gs16_Sevcon2_Debug_MaxFlux				:=	USINT_TO_INT(DebugPMACControl_Rx.au8_Data[0]) +
											SHL(USINT_TO_INT(DebugPMACControl_Rx.au8_Data[1]), 8);
gs16_Sevcon2_Debug_IvLim				:=	USINT_TO_INT(DebugPMACControl_Rx.au8_Data[2]) +
											SHL(USINT_TO_INT(DebugPMACControl_Rx.au8_Data[3]), 8);
gs16_Sevcon2_Debug_IqMax				:=	USINT_TO_INT(DebugPMACControl_Rx.au8_Data[4]) +
											SHL(USINT_TO_INT(DebugPMACControl_Rx.au8_Data[5]), 8);
gs16_Sevcon2_Debug_Ls_Rx				:=	USINT_TO_INT(DebugPMACControl_Rx.au8_Data[6]) +
											SHL(USINT_TO_INT(DebugPMACControl_Rx.au8_Data[7]), 8);

gs16_Sevcon2_Debug_Slip_Rx				:=	USINT_TO_INT(DebugFVControl_Rx.au8_Data[0]) +
											SHL(USINT_TO_INT(DebugFVControl_Rx.au8_Data[1]), 8);
gs16_Sevcon2_Debug_LmSat_Rx				:=	USINT_TO_INT(DebugFVControl_Rx.au8_Data[2]) +
											SHL(USINT_TO_INT(DebugFVControl_Rx.au8_Data[3]), 8);
gs16_Sevcon2_Debug_IqMax2				:=	USINT_TO_INT(DebugFVControl_Rx.au8_Data[4]) +
											SHL(USINT_TO_INT(DebugFVControl_Rx.au8_Data[5]), 8);
gs16_Sevcon2_Debug_RecipFlux			:=	USINT_TO_INT(DebugFVControl_Rx.au8_Data[6]) +
											SHL(USINT_TO_INT(DebugFVControl_Rx.au8_Data[7]), 8);

											
TorqueStatus1_Rx_Timer(IN := NOT(TorqueStatus1_Rx.q_NewData), PT := T#3S);
TorqueStatus2_Rx_Timer(IN := NOT(TorqueStatus2_Rx.q_NewData), PT := T#3S);
TempStatus_Rx_Timer(IN := NOT(TempStatus_Rx.q_NewData), PT := T#3S);
FaultStatus_Rx_Timer(IN := NOT(FaultStatus_Rx.q_NewData), PT := T#3S);
EncoderStatus_Rx_Timer(IN := NOT(EncoderStatus_Rx.q_NewData), PT := T#3S);
DeubgCurrents_Rx_Timer(IN := NOT(DeubgCurrents_Rx.q_NewData), PT := T#3S);
DebugTemps1_Rx_Timer(IN := NOT(DebugTemps1_Rx.q_NewData), PT := T#3S);
DebugTemps2_Rx_Timer(IN := NOT(DebugTemps2_Rx.q_NewData), PT := T#3S);
DebugPMACControl_Rx_Timer(IN := NOT(DebugPMACControl_Rx.q_NewData), PT := T#3S);
DebugFVControl_Rx_Timer(IN := NOT(DebugFVControl_Rx.q_NewData), PT := T#3S);
IF (TorqueStatus1_Rx_Timer.Q = TRUE AND TorqueStatus2_Rx_Timer.Q = TRUE AND TempStatus_Rx_Timer.Q = TRUE AND
	FaultStatus_Rx_Timer.Q = TRUE AND EncoderStatus_Rx_Timer.Q = TRUE AND DeubgCurrents_Rx_Timer.Q = TRUE AND
	DebugTemps1_Rx_Timer.Q = TRUE AND DebugTemps2_Rx_Timer.Q = TRUE AND DebugPMACControl_Rx_Timer.Q = TRUE AND
	DebugFVControl_Rx_Timer.Q = TRUE) THEN
	gq_Sevcon2_CommsLoss	:=	TRUE;
ELSE
	gq_Sevcon2_CommsLoss	:=	FALSE;
END_IF											


Sevcon2_RxConversion();

END_PROGRAM

// Application/UserCode/Sevcon_Compressor/Sevcon2_RxConversion_1
PROGRAM Sevcon2_RxConversion_1
VAR
END_VAR
VAR CONSTANT
	SIXTEENTH_CF	:	REAL	:=	0.0625;
END_VAR




gr_Sevcon2_TorqueMeasured			:=	gs16_Sevcon2_TorqueMeasured_Rx * SIXTEENTH_CF;
gr_Sevcon2_TorqueAvailableForward	:=	gs16_Sevcon2_TorqueAvailableForward_Rx * SIXTEENTH_CF;
gr_Sevcon2_TorqueAvailableReverse	:=	gs16_Sevcon2_TorqueAvailableReverse_Rx * SIXTEENTH_CF;
gr_Sevcon2_DCLink_Voltage			:=	gs16_Sevcon2_DCLink_Voltage_Rx * SIXTEENTH_CF;
gr_Sevcon2_EncoderPosition			:=	LREAL_TO_REAL(gs32_Sevcon2_EncoderPosition_Rx * (1.5287890625 * EXPT(10, -5)));
gr_Sevcon2_Debug_Id_Act				:=	gs16_Sevcon2_Debug_Id_Act_Rx * SIXTEENTH_CF;
gr_Sevcon2_Debug_Iq_Act				:=	gs16_Sevcon2_Debug_Iq_Act_Rx * SIXTEENTH_CF;
gr_Sevcon2_Debug_Id_Ref				:=	gs16_Sevcon2_Debug_Id_Ref_Rx * SIXTEENTH_CF;
gr_Sevcon2_Debug_Iq_Ref				:=	gs16_Sevcon2_Debug_Iq_Ref_Rx * SIXTEENTH_CF;
gr_Sevcon2_Debug_Ls					:=	LREAL_TO_REAL(gs16_Sevcon2_Debug_Ls_Rx * (5.960464477539 * EXPT(10, -8)));
gr_Sevcon2_Debug_Slip				:=	gs16_Sevcon2_Debug_Slip_Rx * SIXTEENTH_CF;
gr_Sevcon2_Debug_LmSat				:=	LREAL_TO_REAL(gs16_Sevcon2_Debug_LmSat_Rx * (1.52587890625 * EXPT(10, -5)));

END_PROGRAM

// Application/UserCode/Sevcon_Compressor/Sevcon2_Tx_1
PROGRAM Sevcon2_Tx_1
VAR
	ht_TorqueDemand1_Tx			:	EPEC_CANVXD.Msg;
	ht_TorqueDemand2_Tx			:	EPEC_CANVXD.Msg;
	ht_BatteryDemand_Tx			:	EPEC_CANVXD.Msg;
	ht_DirectIControlDemand_Tx	:	EPEC_CANVXD.Msg;
	hton_SendTimer				:	TON;
END_VAR

Sevcon2_TxConversion();

ht_TorqueDemand1_Tx.ID		:=	16#191072FA OR EPEC_CANVXD.MASK_29BIT;
ht_TorqueDemand1_Tx.Data[0]	:=	UINT_TO_USINT(gu16_Sevcon2_TorqueRq_Tx);
ht_TorqueDemand1_Tx.Data[1]	:=	UINT_TO_USINT(SHR(gu16_Sevcon2_TorqueRq_Tx, 8));
ht_TorqueDemand1_Tx.Data[2]	:=	UINT_TO_USINT(gu16_Sevcon2_Controlword);
ht_TorqueDemand1_Tx.Data[3]	:=	UINT_TO_USINT(SHR(gu16_Sevcon2_Controlword, 8));
ht_TorqueDemand1_Tx.Data[4]	:=	UINT_TO_USINT(gu16_Sevcon2_TorqueTractionLimit_Tx);
ht_TorqueDemand1_Tx.Data[5]	:=	UINT_TO_USINT(SHR(gu16_Sevcon2_TorqueTractionLimit_Tx, 8));
ht_TorqueDemand1_Tx.Data[6]	:=	gu8_Sevcon2_SEQCommand1;
ht_TorqueDemand1_Tx.Data[7]	:=	gu8_Sevcon2_CSCommand1;
ht_TorqueDemand1_Tx.Len	:=	8;

ht_TorqueDemand2_Tx.ID		:=	16#191172FA OR EPEC_CANVXD.MASK_29BIT;
ht_TorqueDemand2_Tx.Data[0]	:=	UINT_TO_USINT(gu16_Sevcon2_TorqueRegenLimit_Tx);
ht_TorqueDemand2_Tx.Data[1]	:=	UINT_TO_USINT(SHR(gu16_Sevcon2_TorqueRegenLimit_Tx, 8));
ht_TorqueDemand2_Tx.Data[2]	:=	UINT_TO_USINT(gu16_Sevcon2_SpeedLimitForward);
ht_TorqueDemand2_Tx.Data[3]	:=	UINT_TO_USINT(SHR(gu16_Sevcon2_SpeedLimitForward, 8));
ht_TorqueDemand2_Tx.Data[4]	:=	INT_TO_USINT(gs16_Sevcon2_SpeedLimitReverse);
ht_TorqueDemand2_Tx.Data[5]	:=	INT_TO_USINT(SHR(gs16_Sevcon2_SpeedLimitReverse, 8));
ht_TorqueDemand2_Tx.Data[6]	:=	gu8_Sevcon2_SEQCommand2;
ht_TorqueDemand2_Tx.Data[7]	:=	gu8_Sevcon2_CSCommand2;
ht_TorqueDemand2_Tx.Len		:=	8;

ht_BatteryDemand_Tx.ID		:=	16#191272FA OR EPEC_CANVXD.MASK_29BIT;
ht_BatteryDemand_Tx.Data[0]	:=	UINT_TO_USINT(gu16_Sevcon2_DCLink_ImaxDischarge);
ht_BatteryDemand_Tx.Data[1]	:=	UINT_TO_USINT(SHR(gu16_Sevcon2_DCLink_ImaxDischarge, 8));
ht_BatteryDemand_Tx.Data[2]	:=	INT_TO_USINT(gs16_Sevcon2_DCLink_ImaxRecharge);
ht_BatteryDemand_Tx.Data[3]	:=	INT_TO_USINT(SHR(gs16_Sevcon2_DCLink_ImaxRecharge, 8));
ht_BatteryDemand_Tx.Data[4]	:=	UINT_TO_USINT(gu16_Sevcon2_DCLink_VoltageTarget_Tx);
ht_BatteryDemand_Tx.Data[5]	:=	UINT_TO_USINT(SHR(gu16_Sevcon2_DCLink_VoltageTarget_Tx, 8));
ht_BatteryDemand_Tx.Data[6]	:=	gu8_Sevcon1_SEQCurrentLimits;
ht_BatteryDemand_Tx.Data[7]	:=	gu8_Sevcon1_CSCurrentLimits;
ht_BatteryDemand_Tx.Len		:=	8;
	
ht_DirectIControlDemand_Tx.ID		:=	16#191372FA OR EPEC_CANVXD.MASK_29BIT;
ht_DirectIControlDemand_Tx.Data[0]	:=	UINT_TO_USINT(gu16_Sevcon2_DebugIqDirectControl_Tx);
ht_DirectIControlDemand_Tx.Data[1]	:=	UINT_TO_USINT(SHR(gu16_Sevcon2_DebugIqDirectControl_Tx, 8));
ht_DirectIControlDemand_Tx.Data[2]	:=	UINT_TO_USINT(gu16_Sevcon2_DebugIdDirectControl_Tx);
ht_DirectIControlDemand_Tx.Data[3]	:=	UINT_TO_USINT(SHR(gu16_Sevcon2_DebugIdDirectControl_Tx, 8));
ht_DirectIControlDemand_Tx.Data[4]	:=	0;
ht_DirectIControlDemand_Tx.Data[5]	:=	0;
ht_DirectIControlDemand_Tx.Data[6]	:=	gu8_Sevcon1_DirectCurrents;
ht_DirectIControlDemand_Tx.Data[7]	:=	gu8_Sevcon1_CSDirectCurrents;
ht_DirectIControlDemand_Tx.Len		:=	8;
	
hton_SendTimer(IN := TRUE, PT := T#50MS);
IF (hton_SendTimer.Q = TRUE) THEN
	G_CAN2_Channel.SendMessage(i_pMSG:=ADR(ht_TorqueDemand1_Tx));
	G_CAN2_Channel.SendMessage(i_pMSG:=ADR(ht_BatteryDemand_Tx));
	(*G_CAN2_Channel.SendMessage(i_pMSG:=ADR(ht_DirectIControlDemand_Tx));*)
	G_CAN2_Channel.SendMessage(i_pMSG:=ADR(ht_TorqueDemand2_Tx));
	hton_SendTimer(IN := FALSE, PT := T#0MS);
END_IF

END_PROGRAM

// Application/UserCode/Sevcon_Compressor/Sevcon2_TxConversion_1
PROGRAM Sevcon2_TxConversion_1
VAR
END_VAR
VAR CONSTANT
	SEVCON_TX_CF	:	REAL	:=	0.0625;
END_VAR




gu16_Sevcon2_TorqueRq_Tx				:=	REAL_TO_UINT(gr_Sevcon2_TorqueRq / SEVCON_TX_CF);
gu16_Sevcon2_TorqueTractionLimit_Tx		:=	REAL_TO_UINT(gr_Sevcon2_TorqueTractionLimit / SEVCON_TX_CF);
gu16_Sevcon2_TorqueRegenLimit_Tx		:=	REAL_TO_UINT(gr_Sevcon2_TorqueRegenLimit / SEVCON_TX_CF);
gu16_Sevcon2_DCLink_VoltageTarget_Tx	:=	REAL_TO_UINT(gr_Sevcon2_DCLink_VoltageTarget / SEVCON_TX_CF);
gu16_Sevcon2_DebugIqDirectControl_Tx	:=	REAL_TO_UINT(gr_Sevcon2_DebugIqDirectControl / SEVCON_TX_CF);
gu16_Sevcon2_DebugIdDirectControl_Tx	:=	REAL_TO_UINT(gr_Sevcon2_DebugIdDirectControl / SEVCON_TX_CF);

END_PROGRAM

// Application/UserCode/Sevcon ePTO/Sevcon_ePTO_Control
PROGRAM Sevcon_ePTO_Control
VAR_INPUT
	hton_WindUpTorque_Timer	:	TON;
	hq_PowerSteering_Enable	:	BOOL;
	hton_HandbrakeOffTimer	:	TON;
	hr_SteeringSpeed		:	REAL;
END_VAR
VAR_OUTPUT
END_VAR
VAR
	hq_ePTO_Request: BOOL := FALSE;
	hr_ePTO_Speed: INT := 400;
	gq_ePTO_Test: BOOL := FALSE;
END_VAR
VAR CONSTANT
	(*Statuswords*)
	NOTREADY_STAT				:	USINT	:=	1;
	SHUTDOWN_STAT				:	USINT	:=	2;
	PRECHARGE_STAT				:	USINT	:=	4;
	ENERGISED_STAT				:	USINT	:=	7;
	ENABLED_STAT				:	USINT	:=	8;
	FAULTREACTIONACTIVE_STAT	:	USINT	:=	11;
	FAULTOFF_STAT				:	USINT	:=	13;
	ACTIVESHORT_STAT			:	USINT	:=	14;
	(*Commandwords*)
	NOCOMMAND_COMM		:	USINT	:=	0;
	ENERGISE_COMM		:	USINT	:=	3;
	ENABLED_COMM		:	USINT	:=	5;
	SHUTDOWN_COMM		:	USINT	:=	6;
	FAULTRESET_COMM		:	USINT	:=	9;
	ACTIVESHORT_COMM	:	USINT	:=	10;
	
	TORQUE_RQ			:	USINT	:=	200;
	REVERSE_SPD_LIMIT	:	INT		:=	-500;
	MAX_DISCHARGE		:	USINT	:=	50;
	MAX_CHARGE			:	SINT	:=	-50;
	TRACTION_LIMIT		:	USINT	:=	100;
	
	CANBUS_OFF			:	INT	:=	21256;
END_VAR

VAR RETAIN
	ePTO_Speed: INT := 1200;
END_VAR



(**)
(*Check for Comms fault*)
IF (gu8_SystemState = DRIVE_SYS AND DOS_q_BatteryDischargeMain_DO = TRUE) THEN
	IF (gu8_Sevcon_ePTO_InverterStatus = FAULTOFF_STAT OR gu8_Sevcon_ePTO_InverterStatus = ACTIVESHORT_STAT) THEN
		gu16_Sevcon_ePTO_Controlword	:=	FAULTRESET_COMM;
	ELSIF (gu8_Sevcon_ePTO_InverterStatus = NOTREADY_STAT OR gu8_Sevcon_ePTO_InverterStatus = SHUTDOWN_STAT) THEN
		gu16_Sevcon_ePTO_Controlword	:=	ENERGISE_COMM;
	ELSIF (gu8_Sevcon_ePTO_InverterStatus = PRECHARGE_STAT) THEN
		gu16_Sevcon_ePTO_Controlword	:=	ENERGISE_COMM;
	ELSIF (gu8_Sevcon_ePTO_InverterStatus = ENERGISED_STAT) THEN
		gu16_Sevcon_ePTO_Controlword	:=	ENABLED_COMM;
	ELSIF (gu8_Sevcon_ePTO_InverterStatus = ENABLED_STAT) THEN
		gu16_Sevcon_ePTO_Controlword	:=	ENABLED_COMM;
	ELSE
		gu16_Sevcon_ePTO_Controlword	:=	NOCOMMAND_COMM;
	END_IF
ELSE
	gu16_Sevcon_ePTO_Controlword	:=	SHUTDOWN_COMM;
END_IF

(*hton_HandbrakeOffTimer(IN := gq_HandBrake, PT := T#30S);*)
(*This could be changed to link to the current speed of the vehicle in which case the different gear ratios and wheel diameter will be needed here to calculate*)
IF ((gq_ePTO_Test = TRUE OR DI_q_DirectionSwitch_DriveCrawl_DI = TRUE) AND gu8_SystemState = DRIVE_SYS) THEN (*change this to the input to start the body eg. oil request*)
	hq_ePTO_Request	:=	TRUE;
	hr_ePTO_Speed	:=	ePTO_Speed; (*Ensure the speed limit is never set negative*);
	gu16_Sevcon_ePTO_SpeedLimitForward	:=	REAL_TO_UINT(LIMIT(400, hr_ePTO_Speed, 2000)); (*Controlling the speed through the limits*)
	gr_Sevcon_ePTO_TorqueRq						:=	TORQUE_RQ;
ELSIF (gu8_SystemState = DRIVE_SYS) THEN
	hq_ePTO_Request	:=	FALSE;
	gu16_Sevcon_ePTO_SpeedLimitForward	:=	0;
	gr_Sevcon_ePTO_TorqueRq				:=	0;
END_IF



(*All these are constants to be sent out to the Sevcon unit and do not need changing during operation*)
(*IF (gu8_Sevcon_ePTO_InverterStatus = ENABLED_STAT) THEN
	hton_WindUpTorque_Timer(IN := TRUE, PT := T#5000MS);
	gr_Sevcon_ePTO_TorqueRq						:=	TORQUE_RQ * (TIME_TO_REAL(hton_WindUpTorque_Timer.ET) / 5000);
ELSE
	hton_WindUpTorque_Timer(IN := FALSE, PT := T#0MS);
	gr_Sevcon_ePTO_TorqueRq						:=	0;
END_IF*)

gr_Sevcon_ePTO_DCLink_VoltageTarget			:=	0; (*Not needed as not being used as a generator*)
gs16_Sevcon_ePTO_SpeedLimitReverse			:=	REVERSE_SPD_LIMIT;
gu16_Sevcon_ePTO_DCLink_ImaxDischarge		:=	MAX_DISCHARGE;
gs16_Sevcon_ePTO_DCLink_ImaxRecharge		:=	MAX_CHARGE;
gr_Sevcon_ePTO_TorqueTractionLimit			:=	TRACTION_LIMIT;
gr_Sevcon_ePTO_TorqueRegenLimit				:=	0;

gu8_Sevcon_ePTO_CSCommand1					:=	0;
gu8_Sevcon_ePTO_CSCommand2					:=	0;
gu8_Sevcon_ePTO_CSCurrentLimits				:=	0;
(*Counters to run every cycle and increment so the Sevcons know the VMU is still running*)
IF (gu8_Sevcon_ePTO_SEQCommand1 < 255) THEN
	gu8_Sevcon_ePTO_SEQCommand1			:=	gu8_Sevcon_ePTO_SEQCommand1 + 1;
ELSE
	gu8_Sevcon_ePTO_SEQCommand1			:=	0;
END_IF
IF (gu8_Sevcon_ePTO_SEQCommand2 < 255) THEN
	gu8_Sevcon_ePTO_SEQCommand2			:=	gu8_Sevcon_ePTO_SEQCommand2 + 1;
ELSE
	gu8_Sevcon_ePTO_SEQCommand2			:=	0;
END_IF
IF (gu8_Sevcon_ePTO_SEQCurrentLimits < 255) THEN
	gu8_Sevcon_ePTO_SEQCurrentLimits	:=	gu8_Sevcon_ePTO_SEQCurrentLimits + 1;
ELSE
	gu8_Sevcon_ePTO_SEQCurrentLimits	:=	0;
END_IF

END_PROGRAM

// Application/UserCode/Sevcon ePTO/Sevcon_ePTO_Rx
PROGRAM Sevcon_ePTO_Rx
VAR
	TorqueStatus1_Rx	:	Receive_CAN4_EXD;
	TorqueStatus2_Rx	:	Receive_CAN4_EXD;
	TempStatus_Rx		:	Receive_CAN4_EXD;
	FaultStatus_Rx		:	Receive_CAN4_EXD;
	EncoderStatus_Rx	:	Receive_CAN4_EXD;
	DeubgCurrents_Rx	:	Receive_CAN4_EXD;
	DebugTemps1_Rx		:	Receive_CAN4_EXD;
	DebugTemps2_Rx		:	Receive_CAN4_EXD;
	DebugPMACControl_Rx	:	Receive_CAN4_EXD;
	DebugFVControl_Rx	:	Receive_CAN4_EXD;
END_VAR


TorqueStatus1_Rx(u32_COBID	:=	16#1918FF73,
				q_NewData => ,
				au8_Data => ,
				u8_Length => 			);

TorqueStatus2_Rx(u32_COBID	:=	16#1919FF73,
				q_NewData => ,
				au8_Data => ,
				u8_Length => 			);

TempStatus_Rx(u32_COBID	:=	16#191AFF73,
				q_NewData => ,
				au8_Data => ,
				u8_Length => 			);

FaultStatus_Rx(u32_COBID	:=	16#191BFF73,
				q_NewData => ,
				au8_Data => ,
				u8_Length => 			);

EncoderStatus_Rx(u32_COBID	:=	16#191CFF73,
				q_NewData => ,
				au8_Data => ,
				u8_Length => 			);

DeubgCurrents_Rx(u32_COBID	:=	16#1928FF73,
				q_NewData => ,
				au8_Data => ,
				u8_Length => 			);

DebugTemps1_Rx(u32_COBID	:=	16#192AFF73,
				q_NewData => ,
				au8_Data => ,
				u8_Length => 			);

DebugTemps2_Rx(u32_COBID	:=	16#192BFF73,
				q_NewData => ,
				au8_Data => ,
				u8_Length => 			);

DebugPMACControl_Rx(u32_COBID	:=	16#192CFF73,
				q_NewData => ,
				au8_Data => ,
				u8_Length => 			);

DebugFVControl_Rx(u32_COBID	:=	16#192DFF73,
				q_NewData => ,
				au8_Data => ,
				u8_Length => 			);				

			
				
gs16_Sevcon_ePTO_TorqueMeasured_Rx			:=	USINT_TO_INT(TorqueStatus1_Rx.au8_Data[0]) +
											SHL(USINT_TO_INT(TorqueStatus1_Rx.au8_Data[1]), 8);
gs16_Sevcon_ePTO_SpeedMeasured				:=	USINT_TO_INT(TorqueStatus1_Rx.au8_Data[2]) +
											SHL(USINT_TO_INT(TorqueStatus1_Rx.au8_Data[3]), 8);
gs16_Sevcon_ePTO_DCLink_Current				:=	USINT_TO_INT(TorqueStatus1_Rx.au8_Data[4]) +
											SHL(USINT_TO_INT(TorqueStatus1_Rx.au8_Data[5]), 8);
gu8_Sevcon_ePTO_SEQ_Torque					:=	TorqueStatus1_Rx.au8_Data[6];
gu8_Sevcon_ePTO_CS_Torque					:=	TorqueStatus1_Rx.au8_Data[7];

gs16_Sevcon_ePTO_TorqueAvailableForward_Rx	:=	USINT_TO_INT(TorqueStatus2_Rx.au8_Data[0]) +
											SHL(USINT_TO_INT(TorqueStatus2_Rx.au8_Data[1]), 8);
gs16_Sevcon_ePTO_TorqueAvailableReverse_Rx	:=	USINT_TO_INT(TorqueStatus2_Rx.au8_Data[2]) +
											SHL(USINT_TO_INT(TorqueStatus2_Rx.au8_Data[3]), 8);
gu8_Sevcon_ePTO_InverterStatus				:=	TorqueStatus2_Rx.au8_Data[4];
gu8_Sevcon_ePTO_TorqueLimitCode				:=	TorqueStatus2_Rx.au8_Data[5];
gu8_Sevcon_ePTO_SEQ_Status					:=	TorqueStatus2_Rx.au8_Data[6];
gu8_Sevcon_ePTO_CS_Status					:=	TorqueStatus2_Rx.au8_Data[7];

gs16_Sevcon_ePTO_TempRemaining				:=	USINT_TO_INT(TempStatus_Rx.au8_Data[0]) +
											SHL(USINT_TO_INT(TempStatus_Rx.au8_Data[1]), 8);
gs16_Sevcon_ePTO_MotorTemp					:=	USINT_TO_INT(TempStatus_Rx.au8_Data[2]) +
											SHL(USINT_TO_INT(TempStatus_Rx.au8_Data[3]), 8);
gs16_Sevcon_ePTO_DCLink_Voltage_Rx			:=	USINT_TO_INT(TempStatus_Rx.au8_Data[4]) +
											SHL(USINT_TO_INT(TempStatus_Rx.au8_Data[5]), 8);
gu8_Sevcon_ePTO_SEQ_Temp					:=	TempStatus_Rx.au8_Data[6];
gu8_Sevcon_ePTO_CS_Temp						:=	TempStatus_Rx.au8_Data[7];

gs16_Sevcon_ePTO_FaultCode					:=	USINT_TO_INT(FaultStatus_Rx.au8_Data[0]) +
											SHL(USINT_TO_INT(FaultStatus_Rx.au8_Data[1]), 8);
gs32_Sevcon_ePTO_FaultData					:=	USINT_TO_DINT(FaultStatus_Rx.au8_Data[2]) +
											SHL(USINT_TO_DINT(FaultStatus_Rx.au8_Data[3]), 8) +
											SHL(USINT_TO_DINT(FaultStatus_Rx.au8_Data[4]), 16) +
											SHL(USINT_TO_DINT(FaultStatus_Rx.au8_Data[5]), 24);
gu8_Sevcon_ePTO_SEQ_Fault					:=	FaultStatus_Rx.au8_Data[6];
gu8_Sevcon_ePTO_CS_Fault					:=	FaultStatus_Rx.au8_Data[7];

gs32_Sevcon_ePTO_EncoderPosition_Rx			:=	USINT_TO_DINT(EncoderStatus_Rx.au8_Data[0]) +
											SHL(USINT_TO_DINT(EncoderStatus_Rx.au8_Data[1]), 8) +
											SHL(USINT_TO_DINT(EncoderStatus_Rx.au8_Data[2]), 16) +
											SHL(USINT_TO_DINT(EncoderStatus_Rx.au8_Data[3]), 24);

gs16_Sevcon_ePTO_Debug_Id_Act_Rx			:=	USINT_TO_INT(DeubgCurrents_Rx.au8_Data[0]) +
											SHL(USINT_TO_INT(DeubgCurrents_Rx.au8_Data[1]), 8);
gs16_Sevcon_ePTO_Debug_Iq_Act_Rx			:=	USINT_TO_INT(DeubgCurrents_Rx.au8_Data[2]) +
											SHL(USINT_TO_INT(DeubgCurrents_Rx.au8_Data[3]), 8);
gs16_Sevcon_ePTO_Debug_Id_Ref_Rx			:=	USINT_TO_INT(DeubgCurrents_Rx.au8_Data[4]) +
											SHL(USINT_TO_INT(DeubgCurrents_Rx.au8_Data[5]), 8);
gs16_Sevcon_ePTO_Debug_Iq_Ref_Rx			:=	USINT_TO_INT(DeubgCurrents_Rx.au8_Data[6]) +
											SHL(USINT_TO_INT(DeubgCurrents_Rx.au8_Data[7]), 8);

gu8_Sevcon_ePTO_Debug_Temp_Junction0		:=	DebugTemps1_Rx.au8_Data[0];
gu8_Sevcon_ePTO_Debug_Temp_Junction1		:=	DebugTemps1_Rx.au8_Data[1];
gu8_Sevcon_ePTO_Debug_Temp_Junction2		:=	DebugTemps1_Rx.au8_Data[2];
gu8_Sevcon_ePTO_Debug_Temp_Junction3		:=	DebugTemps1_Rx.au8_Data[3];
gu8_Sevcon_ePTO_Debug_Temp_Junction4		:=	DebugTemps1_Rx.au8_Data[4];
gu8_Sevcon_ePTO_Debug_Temp_Junction5		:=	DebugTemps1_Rx.au8_Data[5];
gu8_Sevcon_ePTO_Debug_Temp_MotorMeasured	:=	DebugTemps1_Rx.au8_Data[6];
gu8_Sevcon_ePTO_Debug_Temp_MotorEstimate	:=	DebugTemps1_Rx.au8_Data[7];

gu8_Sevcon_ePTO_Debug_Temp_CapEstimateFast	:=	DebugTemps2_Rx.au8_Data[0];
gu8_Sevcon_ePTO_Debug_Temp_Track			:=	DebugTemps2_Rx.au8_Data[1];
gu8_Sevcon_ePTO_Debug_Temp_CapEstimateSlow	:=	DebugTemps2_Rx.au8_Data[2];
gu8_Sevcon_ePTO_Debug_Temp_Heatsink			:=	DebugTemps2_Rx.au8_Data[3];
gu8_Sevcon_ePTO_Debug_Temp_DeltaTj			:=	DebugTemps2_Rx.au8_Data[4];
gu8_Sevcon_ePTO_Debug_Temp_Normalised		:=	DebugTemps2_Rx.au8_Data[5];
gu8_Sevcon_ePTO_Debug_Temp_Coolant			:=	DebugTemps2_Rx.au8_Data[6];
gu8_Sevcon_ePTO_Debug_Temp_Winding			:=	DebugTemps2_Rx.au8_Data[7];

gs16_Sevcon_ePTO_Debug_MaxFlux				:=	USINT_TO_INT(DebugPMACControl_Rx.au8_Data[0]) +
											SHL(USINT_TO_INT(DebugPMACControl_Rx.au8_Data[1]), 8);
gs16_Sevcon_ePTO_Debug_IvLim				:=	USINT_TO_INT(DebugPMACControl_Rx.au8_Data[2]) +
											SHL(USINT_TO_INT(DebugPMACControl_Rx.au8_Data[3]), 8);
gs16_Sevcon_ePTO_Debug_IqMax				:=	USINT_TO_INT(DebugPMACControl_Rx.au8_Data[4]) +
											SHL(USINT_TO_INT(DebugPMACControl_Rx.au8_Data[5]), 8);
gs16_Sevcon_ePTO_Debug_Ls_Rx				:=	USINT_TO_INT(DebugPMACControl_Rx.au8_Data[6]) +
											SHL(USINT_TO_INT(DebugPMACControl_Rx.au8_Data[7]), 8);

gs16_Sevcon_ePTO_Debug_Slip_Rx				:=	USINT_TO_INT(DebugFVControl_Rx.au8_Data[0]) +
											SHL(USINT_TO_INT(DebugFVControl_Rx.au8_Data[1]), 8);
gs16_Sevcon_ePTO_Debug_LmSat_Rx				:=	USINT_TO_INT(DebugFVControl_Rx.au8_Data[2]) +
											SHL(USINT_TO_INT(DebugFVControl_Rx.au8_Data[3]), 8);
gs16_Sevcon_ePTO_Debug_IqMax2				:=	USINT_TO_INT(DebugFVControl_Rx.au8_Data[4]) +
											SHL(USINT_TO_INT(DebugFVControl_Rx.au8_Data[5]), 8);
gs16_Sevcon_ePTO_Debug_RecipFlux			:=	USINT_TO_INT(DebugFVControl_Rx.au8_Data[6]) +
											SHL(USINT_TO_INT(DebugFVControl_Rx.au8_Data[7]), 8);


											
Sevcon_ePTO_RxConversion();

END_PROGRAM

// Application/UserCode/Sevcon ePTO/Sevcon_ePTO_RxConversion
PROGRAM Sevcon_ePTO_RxConversion
VAR
END_VAR
VAR CONSTANT
	SIXTEENTH_CF	:	REAL	:=	0.0625;
END_VAR




gr_Sevcon_ePTO_TorqueMeasured			:=	gs16_Sevcon_ePTO_TorqueMeasured_Rx * SIXTEENTH_CF;
gr_Sevcon_ePTO_TorqueAvailableForward	:=	gs16_Sevcon_ePTO_TorqueAvailableForward_Rx * SIXTEENTH_CF;
gr_Sevcon_ePTO_TorqueAvailableReverse	:=	gs16_Sevcon_ePTO_TorqueAvailableReverse_Rx * SIXTEENTH_CF;
gr_Sevcon_ePTO_DCLink_Voltage			:=	gs16_Sevcon_ePTO_DCLink_Voltage_Rx * SIXTEENTH_CF;
gr_Sevcon_ePTO_EncoderPosition			:=	LREAL_TO_REAL(gs32_Sevcon_ePTO_EncoderPosition_Rx * (1.5287890625 * EXPT(10, -5)));
gr_Sevcon_ePTO_Debug_Id_Act			:=	gs16_Sevcon_ePTO_Debug_Id_Act_Rx * SIXTEENTH_CF;
gr_Sevcon_ePTO_Debug_Iq_Act			:=	gs16_Sevcon_ePTO_Debug_Iq_Act_Rx * SIXTEENTH_CF;
gr_Sevcon_ePTO_Debug_Id_Ref			:=	gs16_Sevcon_ePTO_Debug_Id_Ref_Rx * SIXTEENTH_CF;
gr_Sevcon_ePTO_Debug_Iq_Ref			:=	gs16_Sevcon_ePTO_Debug_Iq_Ref_Rx * SIXTEENTH_CF;
gr_Sevcon_ePTO_Debug_Ls				:=	LREAL_TO_REAL(gs16_Sevcon_ePTO_Debug_Ls_Rx * (5.960464477539 * EXPT(10, -8)));
gr_Sevcon_ePTO_Debug_Slip				:=	gs16_Sevcon_ePTO_Debug_Slip_Rx * SIXTEENTH_CF;
gr_Sevcon_ePTO_Debug_LmSat				:=	LREAL_TO_REAL(gs16_Sevcon_ePTO_Debug_LmSat_Rx * (1.52587890625 * EXPT(10, -5)));

END_PROGRAM

// Application/UserCode/Sevcon ePTO/Sevcon_ePTO_Tx
PROGRAM Sevcon_ePTO_Tx
VAR
	ht_TorqueDemand1_Tx			:	EPEC_CANVXD.Msg;
	ht_TorqueDemand2_Tx			:	EPEC_CANVXD.Msg;
	ht_BatteryDemand_Tx			:	EPEC_CANVXD.Msg;
	ht_DirectIControlDemand_Tx	:	EPEC_CANVXD.Msg;
	hton_SendTimer				:	TON;
END_VAR

Sevcon_ePTO_TxConversion();

ht_TorqueDemand1_Tx.ID		:=	16#191073FA (*191071FA*) OR EPEC_CANVXD.MASK_29BIT;
ht_TorqueDemand1_Tx.Data[0]	:=	UINT_TO_USINT(gu16_Sevcon_ePTO_TorqueRq_Tx);
ht_TorqueDemand1_Tx.Data[1]	:=	UINT_TO_USINT(SHR(gu16_Sevcon_ePTO_TorqueRq_Tx, 8));
ht_TorqueDemand1_Tx.Data[2]	:=	UINT_TO_USINT(gu16_Sevcon_ePTO_Controlword);
ht_TorqueDemand1_Tx.Data[3]	:=	UINT_TO_USINT(SHR(gu16_Sevcon_ePTO_Controlword, 8));
ht_TorqueDemand1_Tx.Data[4]	:=	UINT_TO_USINT(gu16_Sevcon_ePTO_TorqueTractionLimit_Tx);
ht_TorqueDemand1_Tx.Data[5]	:=	UINT_TO_USINT(SHR(gu16_Sevcon_ePTO_TorqueTractionLimit_Tx, 8));
ht_TorqueDemand1_Tx.Data[6]	:=	gu8_Sevcon_ePTO_SEQCommand1;
ht_TorqueDemand1_Tx.Data[7]	:=	gu8_Sevcon_ePTO_CSCommand1;
ht_TorqueDemand1_Tx.Len	:=	8;

ht_TorqueDemand2_Tx.ID		:=	16#191173FA (*191171FA*) OR EPEC_CANVXD.MASK_29BIT;
ht_TorqueDemand2_Tx.Data[0]	:=	UINT_TO_USINT(gu16_Sevcon_ePTO_TorqueRegenLimit_Tx);
ht_TorqueDemand2_Tx.Data[1]	:=	UINT_TO_USINT(SHR(gu16_Sevcon_ePTO_TorqueRegenLimit_Tx, 8));
ht_TorqueDemand2_Tx.Data[2]	:=	UINT_TO_USINT(gu16_Sevcon_ePTO_SpeedLimitForward);
ht_TorqueDemand2_Tx.Data[3]	:=	UINT_TO_USINT(SHR(gu16_Sevcon_ePTO_SpeedLimitForward, 8));
ht_TorqueDemand2_Tx.Data[4]	:=	INT_TO_USINT(gs16_Sevcon_ePTO_SpeedLimitReverse);
ht_TorqueDemand2_Tx.Data[5]	:=	INT_TO_USINT(SHR(gs16_Sevcon_ePTO_SpeedLimitReverse, 8));
ht_TorqueDemand2_Tx.Data[6]	:=	gu8_Sevcon_ePTO_SEQCommand2;
ht_TorqueDemand2_Tx.Data[7]	:=	gu8_Sevcon_ePTO_CSCommand2;
ht_TorqueDemand2_Tx.Len		:=	8;

ht_BatteryDemand_Tx.ID		:=	16#191273FA (*191271FA*) OR EPEC_CANVXD.MASK_29BIT;
ht_BatteryDemand_Tx.Data[0]	:=	UINT_TO_USINT(gu16_Sevcon_ePTO_DCLink_ImaxDischarge);
ht_BatteryDemand_Tx.Data[1]	:=	UINT_TO_USINT(SHR(gu16_Sevcon_ePTO_DCLink_ImaxDischarge, 8));
ht_BatteryDemand_Tx.Data[2]	:=	INT_TO_USINT(gs16_Sevcon_ePTO_DCLink_ImaxRecharge);
ht_BatteryDemand_Tx.Data[3]	:=	INT_TO_USINT(SHR(gs16_Sevcon_ePTO_DCLink_ImaxRecharge, 8));
ht_BatteryDemand_Tx.Data[4]	:=	UINT_TO_USINT(gu16_Sevcon_ePTO_DCLink_VoltageTarget_Tx);
ht_BatteryDemand_Tx.Data[5]	:=	UINT_TO_USINT(SHR(gu16_Sevcon_ePTO_DCLink_VoltageTarget_Tx, 8));
ht_BatteryDemand_Tx.Data[6]	:=	gu8_Sevcon_ePTO_SEQCurrentLimits;
ht_BatteryDemand_Tx.Data[7]	:=	gu8_Sevcon_ePTO_CSCurrentLimits;
ht_BatteryDemand_Tx.Len		:=	8;
	
ht_DirectIControlDemand_Tx.ID		:=	16#191373FA (*191371FA*) OR EPEC_CANVXD.MASK_29BIT;
ht_DirectIControlDemand_Tx.Data[0]	:=	UINT_TO_USINT(gu16_Sevcon_ePTO_DebugIqDirectControl_Tx);
ht_DirectIControlDemand_Tx.Data[1]	:=	UINT_TO_USINT(SHR(gu16_Sevcon_ePTO_DebugIqDirectControl_Tx, 8));
ht_DirectIControlDemand_Tx.Data[2]	:=	UINT_TO_USINT(gu16_Sevcon_ePTO_DebugIdDirectControl_Tx);
ht_DirectIControlDemand_Tx.Data[3]	:=	UINT_TO_USINT(SHR(gu16_Sevcon_ePTO_DebugIdDirectControl_Tx, 8));
ht_DirectIControlDemand_Tx.Data[4]	:=	0;
ht_DirectIControlDemand_Tx.Data[5]	:=	0;
ht_DirectIControlDemand_Tx.Data[6]	:=	gu8_Sevcon_ePTO_DirectCurrents;
ht_DirectIControlDemand_Tx.Data[7]	:=	gu8_Sevcon_ePTO_CSDirectCurrents;
ht_DirectIControlDemand_Tx.Len		:=	8;
	
hton_SendTimer(IN := TRUE, PT := T#50MS);
IF (hton_SendTimer.Q = TRUE) THEN
	G_CAN4_Channel.SendMessage(i_pMSG:=ADR(ht_TorqueDemand1_Tx));
	G_CAN4_Channel.SendMessage(i_pMSG:=ADR(ht_BatteryDemand_Tx));
	G_CAN4_Channel.SendMessage(i_pMSG:=ADR(ht_DirectIControlDemand_Tx));
	G_CAN4_Channel.SendMessage(i_pMSG:=ADR(ht_TorqueDemand2_Tx));
	hton_SendTimer(IN := FALSE, PT := T#0MS);
END_IF

END_PROGRAM

// Application/UserCode/Sevcon ePTO/Sevcon_ePTO_TxConversion
PROGRAM Sevcon_ePTO_TxConversion
VAR
END_VAR
VAR CONSTANT
	SEVCON_TX_CF	:	REAL	:=	0.0625;
END_VAR




gu16_Sevcon_ePTO_TorqueRq_Tx				:=	REAL_TO_UINT(gr_Sevcon_ePTO_TorqueRq / SEVCON_TX_CF);
gu16_Sevcon_ePTO_TorqueTractionLimit_Tx		:=	REAL_TO_UINT(gr_Sevcon_ePTO_TorqueTractionLimit / SEVCON_TX_CF);
gu16_Sevcon_ePTO_TorqueRegenLimit_Tx		:=	REAL_TO_UINT(gr_Sevcon_ePTO_TorqueRegenLimit / SEVCON_TX_CF);
gu16_Sevcon_ePTO_DCLink_VoltageTarget_Tx	:=	REAL_TO_UINT(gr_Sevcon_ePTO_DCLink_VoltageTarget / SEVCON_TX_CF);
gu16_Sevcon_ePTO_DebugIqDirectControl_Tx	:=	REAL_TO_UINT(gr_Sevcon_ePTO_DebugIqDirectControl / SEVCON_TX_CF);
gu16_Sevcon_ePTO_DebugIdDirectControl_Tx	:=	REAL_TO_UINT(gr_Sevcon_ePTO_DebugIdDirectControl / SEVCON_TX_CF);

END_PROGRAM

// Application/UserCode/Sevcon_PSP/Sevcon_Steer_Control_1
PROGRAM Sevcon_Steer_Control_1
VAR
	hton_WindUpTorque_Timer	:	TON;
	hq_PowerSteering_Enable	:	BOOL;
	hton_HandbrakeOffTimer	:	TON;
	hr_SteeringSpeed		:	REAL;
	hton_PowerSteeringOff	:	TON;
	Steering_Speed_Setpoint: INT := 2200; //changed from 2000
END_VAR
VAR CONSTANT
	(*Statuswords*)
	NOTREADY_STAT				:	USINT	:=	1;
	SHUTDOWN_STAT				:	USINT	:=	2;
	PRECHARGE_STAT				:	USINT	:=	4;
	ENERGISED_STAT				:	USINT	:=	7;
	ENABLED_STAT				:	USINT	:=	8;
	FAULTREACTIONACTIVE_STAT	:	USINT	:=	11;
	FAULTOFF_STAT				:	USINT	:=	13;
	ACTIVESHORT_STAT			:	USINT	:=	14;
	(*Commandwords*)
	NOCOMMAND_COMM		:	USINT	:=	0;
	ENERGISE_COMM		:	USINT	:=	3;
	ENABLED_COMM		:	USINT	:=	5;
	SHUTDOWN_COMM		:	USINT	:=	6;
	FAULTRESET_COMM		:	USINT	:=	9;
	ACTIVESHORT_COMM	:	USINT	:=	10;
	
	TORQUE_RQ			:	USINT	:=	200;
	REVERSE_SPD_LIMIT	:	INT		:=	-500;
	MAX_DISCHARGE		:	USINT	:=	50;
	MAX_CHARGE			:	SINT	:=	-50;
	TRACTION_LIMIT		:	USINT	:=	100;
	
	CANBUS_OFF			:	INT	:=	21256;
END_VAR


(**)
(*Check for Comms fault*)
IF (gu8_SystemState = DRIVE_SYS AND DOS_q_BatteryDischargeMain_DO = TRUE) THEN
	DO_q_DrievtrainPowerSteering_DO	:=	TRUE;
	IF (gu8_Sevcon1_InverterStatus = FAULTOFF_STAT OR gu8_Sevcon1_InverterStatus = ACTIVESHORT_STAT) THEN
		gu16_Sevcon1_Controlword	:=	FAULTRESET_COMM;
	ELSIF (gu8_Sevcon1_InverterStatus = NOTREADY_STAT OR gu8_Sevcon1_InverterStatus = SHUTDOWN_STAT) THEN
		gu16_Sevcon1_Controlword	:=	ENERGISE_COMM;
	ELSIF (gu8_Sevcon1_InverterStatus = PRECHARGE_STAT) THEN
		gu16_Sevcon1_Controlword	:=	ENERGISE_COMM;
	ELSIF (gu8_Sevcon1_InverterStatus = ENERGISED_STAT) THEN
		gu16_Sevcon1_Controlword	:=	ENABLED_COMM;
	ELSIF (gu8_Sevcon1_InverterStatus = ENABLED_STAT) THEN
		gu16_Sevcon1_Controlword	:=	ENABLED_COMM;
	ELSE
		gu16_Sevcon1_Controlword	:=	NOCOMMAND_COMM;
	END_IF
ELSE
	DO_q_DrievtrainPowerSteering_DO	:=	FALSE;
	gu16_Sevcon1_Controlword	:=	SHUTDOWN_COMM;
END_IF

hton_HandbrakeOffTimer(IN := HMI_Rx.Hand_Brake_On, PT := T#10MS); //Time changed from 30s to 10ms

(*This could be changed to link to the current speed of the vehicle in which case the different gear ratios and wheel diameter will be needed here to calculate*)
IF ((HMI_Rx.Hand_Brake_On = FALSE OR NOT gq_Gear_Neutral) AND gu8_SystemState = DRIVE_SYS) THEN //TEST FIRST THEN REMOVE THIS COMMENT OR NOT gq_Gear_Neutral
	hq_PowerSteering_Enable	:=	TRUE;
	hr_SteeringSpeed		:=	MAX(REAL_TO_INT(Steering_Speed_Setpoint - (ABS(gr_VehicleSpeed_kmph) * 10)), 0) (*Ensure the speed limit is never set negative*);
	gu16_Sevcon1_SpeedLimitForward	:=	REAL_TO_UINT(LIMIT(200, hr_SteeringSpeed, Steering_Speed_Setpoint)); (*Controlling the speed through the limits*)
	hton_PowerSteeringOff(IN := FALSE, PT := T#0S);
ELSIF ((hton_HandbrakeOffTimer.Q = TRUE AND ABS(gr_VehicleSpeed_kmph) < 3) AND gu8_SystemState = DRIVE_SYS) THEN //AND before DRIVE_SYS changed from OR
	hq_PowerSteering_Enable	:=	FALSE;
	hton_PowerSteeringOff(IN := TRUE, PT := T#10MS);
	
	IF (hton_PowerSteeringOff.Q = TRUE) THEN
		gu16_Sevcon1_SpeedLimitForward	:=	200; //instead of shutting off reduce speed to a minimum
	ELSE
		gu16_Sevcon1_SpeedLimitForward	:=	650;
	END_IF
	
END_IF


(*All these are constants to be sent out to the Sevcon unit and do not need changing during operation*)
IF (gu8_Sevcon1_InverterStatus = ENABLED_STAT) THEN
	hton_WindUpTorque_Timer(IN := TRUE, PT := T#5000MS);
	gr_Sevcon1_TorqueRq						:=	TORQUE_RQ * (TIME_TO_REAL(hton_WindUpTorque_Timer.ET) / 5000);
ELSE
	hton_WindUpTorque_Timer(IN := FALSE, PT := T#0MS);
	gr_Sevcon1_TorqueRq						:=	0;
END_IF

gr_Sevcon1_DCLink_VoltageTarget			:=	0; (*Not needed as not being used as a generator*)
gs16_Sevcon1_SpeedLimitReverse			:=	REVERSE_SPD_LIMIT;
gu16_Sevcon1_DCLink_ImaxDischarge		:=	MAX_DISCHARGE;
gs16_Sevcon1_DCLink_ImaxRecharge		:=	MAX_CHARGE;
gr_Sevcon1_TorqueTractionLimit			:=	TRACTION_LIMIT;
gr_Sevcon1_TorqueRegenLimit				:=	0;

gu8_Sevcon1_CSCommand1					:=	0;
gu8_Sevcon1_CSCommand2					:=	0;
gu8_Sevcon1_CSCurrentLimits				:=	0;

(*Counters to run every cycle and increment so the Sevcons know the VMU is still running*)
IF (gu8_Sevcon1_SEQCommand1 < 255) THEN
	gu8_Sevcon1_SEQCommand1			:=	gu8_Sevcon1_SEQCommand1 + 1;
ELSE
	gu8_Sevcon1_SEQCommand1			:=	0;
END_IF
IF (gu8_Sevcon1_SEQCommand2 < 255) THEN
	gu8_Sevcon1_SEQCommand2			:=	gu8_Sevcon1_SEQCommand2 + 1;
ELSE
	gu8_Sevcon1_SEQCommand2			:=	0;
END_IF
IF (gu8_Sevcon1_SEQCurrentLimits < 255) THEN
	gu8_Sevcon1_SEQCurrentLimits	:=	gu8_Sevcon1_SEQCurrentLimits + 1;
ELSE
	gu8_Sevcon1_SEQCurrentLimits	:=	0;
END_IF

(*Backup Pump*)
IF (hq_PowerSteering_Enable = TRUE AND gs16_Sevcon1_FaultCode = CANBUS_OFF) THEN (* Matt, does something else need ORed*)
	DO_q_BackupPump_DO	:=	TRUE;
	(*Fault state will set from the sevcon error*)
ELSE
	DO_q_BackupPump_DO	:=	FALSE;
END_IF

END_PROGRAM

// Application/UserCode/Sevcon_PSP/Sevcon_Steer_Rx_1
PROGRAM Sevcon_Steer_Rx_1
VAR
	TorqueStatus1_Rx	:	Receive_CAN2_EXD;
	TorqueStatus2_Rx	:	Receive_CAN2_EXD;
	TempStatus_Rx		:	Receive_CAN2_EXD;
	FaultStatus_Rx		:	Receive_CAN2_EXD;
	EncoderStatus_Rx	:	Receive_CAN2_EXD;
	DeubgCurrents_Rx	:	Receive_CAN2_EXD;
	DebugTemps1_Rx		:	Receive_CAN2_EXD;
	DebugTemps2_Rx		:	Receive_CAN2_EXD;
	DebugPMACControl_Rx	:	Receive_CAN2_EXD;
	DebugFVControl_Rx	:	Receive_CAN2_EXD;
	
	TorqueStatus1_Rx_Timer		:	TON;
	TorqueStatus2_Rx_Timer		:	TON;
	TempStatus_Rx_Timer			:	TON;
	FaultStatus_Rx_Timer		:	TON;
	EncoderStatus_Rx_Timer		:	TON;
	DeubgCurrents_Rx_Timer		:	TON;
	DebugTemps1_Rx_Timer		:	TON;
	DebugTemps2_Rx_Timer		:	TON;
	DebugPMACControl_Rx_Timer	:	TON;
	DebugFVControl_Rx_Timer		:	TON;
END_VAR


TorqueStatus1_Rx(u32_COBID	:=	16#1918FF71,
				q_NewData => ,
				au8_Data => ,
				u8_Length => 			);

TorqueStatus2_Rx(u32_COBID	:=	16#1919FF71,
				q_NewData => ,
				au8_Data => ,
				u8_Length => 			);

TempStatus_Rx(u32_COBID	:=	16#191AFF71,
				q_NewData => ,
				au8_Data => ,
				u8_Length => 			);

FaultStatus_Rx(u32_COBID	:=	16#191BFF71,
				q_NewData => ,
				au8_Data => ,
				u8_Length => 			);

EncoderStatus_Rx(u32_COBID	:=	16#191CFF71,
				q_NewData => ,
				au8_Data => ,
				u8_Length => 			);

DeubgCurrents_Rx(u32_COBID	:=	16#1928FF71,
				q_NewData => ,
				au8_Data => ,
				u8_Length => 			);

DebugTemps1_Rx(u32_COBID	:=	16#192AFF71,
				q_NewData => ,
				au8_Data => ,
				u8_Length => 			);

DebugTemps2_Rx(u32_COBID	:=	16#192BFF71,
				q_NewData => ,
				au8_Data => ,
				u8_Length => 			);

DebugPMACControl_Rx(u32_COBID	:=	16#192CFF71,
				q_NewData => ,
				au8_Data => ,
				u8_Length => 			);

DebugFVControl_Rx(u32_COBID	:=	16#192DFF71,
				q_NewData => ,
				au8_Data => ,
				u8_Length => 			);				

			
				
gs16_Sevcon1_TorqueMeasured_Rx			:=	USINT_TO_INT(TorqueStatus1_Rx.au8_Data[0]) +
											SHL(USINT_TO_INT(TorqueStatus1_Rx.au8_Data[1]), 8);
gs16_Sevcon1_SpeedMeasured				:=	USINT_TO_INT(TorqueStatus1_Rx.au8_Data[2]) +
											SHL(USINT_TO_INT(TorqueStatus1_Rx.au8_Data[3]), 8);
gs16_Sevcon1_DCLink_Current				:=	USINT_TO_INT(TorqueStatus1_Rx.au8_Data[4]) +
											SHL(USINT_TO_INT(TorqueStatus1_Rx.au8_Data[5]), 8);
gu8_Sevcon1_SEQ_Torque					:=	TorqueStatus1_Rx.au8_Data[6];
gu8_Sevcon1_CS_Torque					:=	TorqueStatus1_Rx.au8_Data[7];

gs16_Sevcon1_TorqueAvailableForward_Rx	:=	USINT_TO_INT(TorqueStatus2_Rx.au8_Data[0]) +
											SHL(USINT_TO_INT(TorqueStatus2_Rx.au8_Data[1]), 8);
gs16_Sevcon1_TorqueAvailableReverse_Rx	:=	USINT_TO_INT(TorqueStatus2_Rx.au8_Data[2]) +
											SHL(USINT_TO_INT(TorqueStatus2_Rx.au8_Data[3]), 8);
gu8_Sevcon1_InverterStatus				:=	TorqueStatus2_Rx.au8_Data[4];
gu8_Sevcon1_TorqueLimitCode				:=	TorqueStatus2_Rx.au8_Data[5];
gu8_Sevcon1_SEQ_Status					:=	TorqueStatus2_Rx.au8_Data[6];
gu8_Sevcon1_CS_Status					:=	TorqueStatus2_Rx.au8_Data[7];

gs16_Sevcon1_TempRemaining				:=	USINT_TO_INT(TempStatus_Rx.au8_Data[0]) +
											SHL(USINT_TO_INT(TempStatus_Rx.au8_Data[1]), 8);
gs16_Sevcon1_MotorTemp					:=	USINT_TO_INT(TempStatus_Rx.au8_Data[2]) +
											SHL(USINT_TO_INT(TempStatus_Rx.au8_Data[3]), 8);
gs16_Sevcon1_DCLink_Voltage_Rx			:=	USINT_TO_INT(TempStatus_Rx.au8_Data[4]) +
											SHL(USINT_TO_INT(TempStatus_Rx.au8_Data[5]), 8);
gu8_Sevcon1_SEQ_Temp					:=	TempStatus_Rx.au8_Data[6];
gu8_Sevcon1_CS_Temp						:=	TempStatus_Rx.au8_Data[7];

gs16_Sevcon1_FaultCode					:=	USINT_TO_INT(FaultStatus_Rx.au8_Data[0]) +
											SHL(USINT_TO_INT(FaultStatus_Rx.au8_Data[1]), 8);
gs32_Sevcon1_FaultData					:=	USINT_TO_DINT(FaultStatus_Rx.au8_Data[2]) +
											SHL(USINT_TO_DINT(FaultStatus_Rx.au8_Data[3]), 8) +
											SHL(USINT_TO_DINT(FaultStatus_Rx.au8_Data[4]), 16) +
											SHL(USINT_TO_DINT(FaultStatus_Rx.au8_Data[5]), 24);
gu8_Sevcon1_SEQ_Fault					:=	FaultStatus_Rx.au8_Data[6];
gu8_Sevcon1_CS_Fault					:=	FaultStatus_Rx.au8_Data[7];

gs32_Sevcon1_EncoderPosition_Rx			:=	USINT_TO_DINT(EncoderStatus_Rx.au8_Data[0]) +
											SHL(USINT_TO_DINT(EncoderStatus_Rx.au8_Data[1]), 8) +
											SHL(USINT_TO_DINT(EncoderStatus_Rx.au8_Data[2]), 16) +
											SHL(USINT_TO_DINT(EncoderStatus_Rx.au8_Data[3]), 24);

gs16_Sevcon1_Debug_Id_Act_Rx			:=	USINT_TO_INT(DeubgCurrents_Rx.au8_Data[0]) +
											SHL(USINT_TO_INT(DeubgCurrents_Rx.au8_Data[1]), 8);
gs16_Sevcon1_Debug_Iq_Act_Rx			:=	USINT_TO_INT(DeubgCurrents_Rx.au8_Data[2]) +
											SHL(USINT_TO_INT(DeubgCurrents_Rx.au8_Data[3]), 8);
gs16_Sevcon1_Debug_Id_Ref_Rx			:=	USINT_TO_INT(DeubgCurrents_Rx.au8_Data[4]) +
											SHL(USINT_TO_INT(DeubgCurrents_Rx.au8_Data[5]), 8);
gs16_Sevcon1_Debug_Iq_Ref_Rx			:=	USINT_TO_INT(DeubgCurrents_Rx.au8_Data[6]) +
											SHL(USINT_TO_INT(DeubgCurrents_Rx.au8_Data[7]), 8);

gu8_Sevcon1_Debug_Temp_Junction0		:=	DebugTemps1_Rx.au8_Data[0];
gu8_Sevcon1_Debug_Temp_Junction1		:=	DebugTemps1_Rx.au8_Data[1];
gu8_Sevcon1_Debug_Temp_Junction2		:=	DebugTemps1_Rx.au8_Data[2];
gu8_Sevcon1_Debug_Temp_Junction3		:=	DebugTemps1_Rx.au8_Data[3];
gu8_Sevcon1_Debug_Temp_Junction4		:=	DebugTemps1_Rx.au8_Data[4];
gu8_Sevcon1_Debug_Temp_Junction5		:=	DebugTemps1_Rx.au8_Data[5];
gu8_Sevcon1_Debug_Temp_MotorMeasured	:=	DebugTemps1_Rx.au8_Data[6];
gu8_Sevcon1_Debug_Temp_MotorEstimate	:=	DebugTemps1_Rx.au8_Data[7];

gu8_Sevcon1_Debug_Temp_CapEstimateFast	:=	DebugTemps2_Rx.au8_Data[0];
gu8_Sevcon1_Debug_Temp_Track			:=	DebugTemps2_Rx.au8_Data[1];
gu8_Sevcon1_Debug_Temp_CapEstimateSlow	:=	DebugTemps2_Rx.au8_Data[2];
gu8_Sevcon1_Debug_Temp_Heatsink			:=	DebugTemps2_Rx.au8_Data[3];
gu8_Sevcon1_Debug_Temp_DeltaTj			:=	DebugTemps2_Rx.au8_Data[4];
gu8_Sevcon1_Debug_Temp_Normalised		:=	DebugTemps2_Rx.au8_Data[5];
gu8_Sevcon1_Debug_Temp_Coolant			:=	DebugTemps2_Rx.au8_Data[6];
gu8_Sevcon1_Debug_Temp_Winding			:=	DebugTemps2_Rx.au8_Data[7];

gs16_Sevcon1_Debug_MaxFlux				:=	USINT_TO_INT(DebugPMACControl_Rx.au8_Data[0]) +
											SHL(USINT_TO_INT(DebugPMACControl_Rx.au8_Data[1]), 8);
gs16_Sevcon1_Debug_IvLim				:=	USINT_TO_INT(DebugPMACControl_Rx.au8_Data[2]) +
											SHL(USINT_TO_INT(DebugPMACControl_Rx.au8_Data[3]), 8);
gs16_Sevcon1_Debug_IqMax				:=	USINT_TO_INT(DebugPMACControl_Rx.au8_Data[4]) +
											SHL(USINT_TO_INT(DebugPMACControl_Rx.au8_Data[5]), 8);
gs16_Sevcon1_Debug_Ls_Rx				:=	USINT_TO_INT(DebugPMACControl_Rx.au8_Data[6]) +
											SHL(USINT_TO_INT(DebugPMACControl_Rx.au8_Data[7]), 8);

gs16_Sevcon1_Debug_Slip_Rx				:=	USINT_TO_INT(DebugFVControl_Rx.au8_Data[0]) +
											SHL(USINT_TO_INT(DebugFVControl_Rx.au8_Data[1]), 8);
gs16_Sevcon1_Debug_LmSat_Rx				:=	USINT_TO_INT(DebugFVControl_Rx.au8_Data[2]) +
											SHL(USINT_TO_INT(DebugFVControl_Rx.au8_Data[3]), 8);
gs16_Sevcon1_Debug_IqMax2				:=	USINT_TO_INT(DebugFVControl_Rx.au8_Data[4]) +
											SHL(USINT_TO_INT(DebugFVControl_Rx.au8_Data[5]), 8);
gs16_Sevcon1_Debug_RecipFlux			:=	USINT_TO_INT(DebugFVControl_Rx.au8_Data[6]) +
											SHL(USINT_TO_INT(DebugFVControl_Rx.au8_Data[7]), 8);


TorqueStatus1_Rx_Timer(IN := NOT(TorqueStatus1_Rx.q_NewData), PT := T#3S);
TorqueStatus2_Rx_Timer(IN := NOT(TorqueStatus2_Rx.q_NewData), PT := T#3S);
TempStatus_Rx_Timer(IN := NOT(TempStatus_Rx.q_NewData), PT := T#3S);
FaultStatus_Rx_Timer(IN := NOT(FaultStatus_Rx.q_NewData), PT := T#3S);
EncoderStatus_Rx_Timer(IN := NOT(EncoderStatus_Rx.q_NewData), PT := T#3S);
DeubgCurrents_Rx_Timer(IN := NOT(DeubgCurrents_Rx.q_NewData), PT := T#3S);
DebugTemps1_Rx_Timer(IN := NOT(DebugTemps1_Rx.q_NewData), PT := T#3S);
DebugTemps2_Rx_Timer(IN := NOT(DebugTemps2_Rx.q_NewData), PT := T#3S);
DebugPMACControl_Rx_Timer(IN := NOT(DebugPMACControl_Rx.q_NewData), PT := T#3S);
DebugFVControl_Rx_Timer(IN := NOT(DebugFVControl_Rx.q_NewData), PT := T#3S);
IF (TorqueStatus1_Rx_Timer.Q = TRUE AND TorqueStatus2_Rx_Timer.Q = TRUE AND TempStatus_Rx_Timer.Q = TRUE AND
	FaultStatus_Rx_Timer.Q = TRUE AND EncoderStatus_Rx_Timer.Q = TRUE AND DeubgCurrents_Rx_Timer.Q = TRUE AND
	DebugTemps1_Rx_Timer.Q = TRUE AND DebugTemps2_Rx_Timer.Q = TRUE AND DebugPMACControl_Rx_Timer.Q = TRUE AND
	DebugFVControl_Rx_Timer.Q = TRUE) THEN
	gq_Sevcon1_CommsLoss	:=	TRUE;
ELSE
	gq_Sevcon1_CommsLoss	:=	FALSE;
END_IF
										
Sevcon_Steer_RxConversion();

END_PROGRAM

// Application/UserCode/Sevcon_PSP/Sevcon_Steer_RxConversion_1
PROGRAM Sevcon_Steer_RxConversion_1
VAR
END_VAR
VAR CONSTANT
	SIXTEENTH_CF	:	REAL	:=	0.0625;
END_VAR




gr_Sevcon1_TorqueMeasured			:=	gs16_Sevcon1_TorqueMeasured_Rx * SIXTEENTH_CF;
gr_Sevcon1_TorqueAvailableForward	:=	gs16_Sevcon1_TorqueAvailableForward_Rx * SIXTEENTH_CF;
gr_Sevcon1_TorqueAvailableReverse	:=	gs16_Sevcon1_TorqueAvailableReverse_Rx * SIXTEENTH_CF;
gr_Sevcon1_DCLink_Voltage			:=	gs16_Sevcon1_DCLink_Voltage_Rx * SIXTEENTH_CF;
gr_Sevcon1_EncoderPosition			:=	LREAL_TO_REAL(gs32_Sevcon1_EncoderPosition_Rx * (1.5287890625 * EXPT(10, -5)));
gr_Sevcon1_Debug_Id_Act				:=	gs16_Sevcon1_Debug_Id_Act_Rx * SIXTEENTH_CF;
gr_Sevcon1_Debug_Iq_Act				:=	gs16_Sevcon1_Debug_Iq_Act_Rx * SIXTEENTH_CF;
gr_Sevcon1_Debug_Id_Ref				:=	gs16_Sevcon1_Debug_Id_Ref_Rx * SIXTEENTH_CF;
gr_Sevcon1_Debug_Iq_Ref				:=	gs16_Sevcon1_Debug_Iq_Ref_Rx * SIXTEENTH_CF;
gr_Sevcon1_Debug_Ls					:=	LREAL_TO_REAL(gs16_Sevcon1_Debug_Ls_Rx * (5.960464477539 * EXPT(10, -8)));
gr_Sevcon1_Debug_Slip				:=	gs16_Sevcon1_Debug_Slip_Rx * SIXTEENTH_CF;
gr_Sevcon1_Debug_LmSat				:=	LREAL_TO_REAL(gs16_Sevcon1_Debug_LmSat_Rx * (1.52587890625 * EXPT(10, -5)));

END_PROGRAM

// Application/UserCode/Sevcon_PSP/Sevcon_Steer_Tx_1
PROGRAM Sevcon_Steer_Tx_1
VAR
	ht_TorqueDemand1_Tx			:	EPEC_CANVXD.Msg;
	ht_TorqueDemand2_Tx			:	EPEC_CANVXD.Msg;
	ht_BatteryDemand_Tx			:	EPEC_CANVXD.Msg;
	ht_DirectIControlDemand_Tx	:	EPEC_CANVXD.Msg;
	hton_SendTimer				:	TON;
END_VAR

Sevcon_Steer_TxConversion();

ht_TorqueDemand1_Tx.ID		:=	16#191071FA OR EPEC_CANVXD.MASK_29BIT;
ht_TorqueDemand1_Tx.Data[0]	:=	UINT_TO_USINT(gu16_Sevcon1_TorqueRq_Tx);
ht_TorqueDemand1_Tx.Data[1]	:=	UINT_TO_USINT(SHR(gu16_Sevcon1_TorqueRq_Tx, 8));
ht_TorqueDemand1_Tx.Data[2]	:=	UINT_TO_USINT(gu16_Sevcon1_Controlword);
ht_TorqueDemand1_Tx.Data[3]	:=	UINT_TO_USINT(SHR(gu16_Sevcon1_Controlword, 8));
ht_TorqueDemand1_Tx.Data[4]	:=	UINT_TO_USINT(gu16_Sevcon1_TorqueTractionLimit_Tx);
ht_TorqueDemand1_Tx.Data[5]	:=	UINT_TO_USINT(SHR(gu16_Sevcon1_TorqueTractionLimit_Tx, 8));
ht_TorqueDemand1_Tx.Data[6]	:=	gu8_Sevcon1_SEQCommand1;
ht_TorqueDemand1_Tx.Data[7]	:=	gu8_Sevcon1_CSCommand1;
ht_TorqueDemand1_Tx.Len	:=	8;

ht_TorqueDemand2_Tx.ID		:=	16#191171FA OR EPEC_CANVXD.MASK_29BIT;
ht_TorqueDemand2_Tx.Data[0]	:=	UINT_TO_USINT(gu16_Sevcon1_TorqueRegenLimit_Tx);
ht_TorqueDemand2_Tx.Data[1]	:=	UINT_TO_USINT(SHR(gu16_Sevcon1_TorqueRegenLimit_Tx, 8));
ht_TorqueDemand2_Tx.Data[2]	:=	UINT_TO_USINT(gu16_Sevcon1_SpeedLimitForward);
ht_TorqueDemand2_Tx.Data[3]	:=	UINT_TO_USINT(SHR(gu16_Sevcon1_SpeedLimitForward, 8));
ht_TorqueDemand2_Tx.Data[4]	:=	INT_TO_USINT(gs16_Sevcon1_SpeedLimitReverse);
ht_TorqueDemand2_Tx.Data[5]	:=	INT_TO_USINT(SHR(gs16_Sevcon1_SpeedLimitReverse, 8));
ht_TorqueDemand2_Tx.Data[6]	:=	gu8_Sevcon1_SEQCommand2;
ht_TorqueDemand2_Tx.Data[7]	:=	gu8_Sevcon1_CSCommand2;
ht_TorqueDemand2_Tx.Len		:=	8;

ht_BatteryDemand_Tx.ID		:=	16#191271FA OR EPEC_CANVXD.MASK_29BIT;
ht_BatteryDemand_Tx.Data[0]	:=	UINT_TO_USINT(gu16_Sevcon1_DCLink_ImaxDischarge);
ht_BatteryDemand_Tx.Data[1]	:=	UINT_TO_USINT(SHR(gu16_Sevcon1_DCLink_ImaxDischarge, 8));
ht_BatteryDemand_Tx.Data[2]	:=	INT_TO_USINT(gs16_Sevcon1_DCLink_ImaxRecharge);
ht_BatteryDemand_Tx.Data[3]	:=	INT_TO_USINT(SHR(gs16_Sevcon1_DCLink_ImaxRecharge, 8));
ht_BatteryDemand_Tx.Data[4]	:=	UINT_TO_USINT(gu16_Sevcon1_DCLink_VoltageTarget_Tx);
ht_BatteryDemand_Tx.Data[5]	:=	UINT_TO_USINT(SHR(gu16_Sevcon1_DCLink_VoltageTarget_Tx, 8));
ht_BatteryDemand_Tx.Data[6]	:=	gu8_Sevcon1_SEQCurrentLimits;
ht_BatteryDemand_Tx.Data[7]	:=	gu8_Sevcon1_CSCurrentLimits;
ht_BatteryDemand_Tx.Len		:=	8;
	
ht_DirectIControlDemand_Tx.ID		:=	16#191371FA OR EPEC_CANVXD.MASK_29BIT;
ht_DirectIControlDemand_Tx.Data[0]	:=	UINT_TO_USINT(gu16_Sevcon1_DebugIqDirectControl_Tx);
ht_DirectIControlDemand_Tx.Data[1]	:=	UINT_TO_USINT(SHR(gu16_Sevcon1_DebugIqDirectControl_Tx, 8));
ht_DirectIControlDemand_Tx.Data[2]	:=	UINT_TO_USINT(gu16_Sevcon1_DebugIdDirectControl_Tx);
ht_DirectIControlDemand_Tx.Data[3]	:=	UINT_TO_USINT(SHR(gu16_Sevcon1_DebugIdDirectControl_Tx, 8));
ht_DirectIControlDemand_Tx.Data[4]	:=	0;
ht_DirectIControlDemand_Tx.Data[5]	:=	0;
ht_DirectIControlDemand_Tx.Data[6]	:=	gu8_Sevcon1_DirectCurrents;
ht_DirectIControlDemand_Tx.Data[7]	:=	gu8_Sevcon1_CSDirectCurrents;
ht_DirectIControlDemand_Tx.Len		:=	8;
	
hton_SendTimer(IN := TRUE, PT := T#50MS);
IF (hton_SendTimer.Q = TRUE) THEN
	G_CAN2_Channel.SendMessage(i_pMSG:=ADR(ht_TorqueDemand1_Tx));
	G_CAN2_Channel.SendMessage(i_pMSG:=ADR(ht_BatteryDemand_Tx));
	G_CAN2_Channel.SendMessage(i_pMSG:=ADR(ht_DirectIControlDemand_Tx));
	G_CAN2_Channel.SendMessage(i_pMSG:=ADR(ht_TorqueDemand2_Tx));
	hton_SendTimer(IN := FALSE, PT := T#0MS);
END_IF

END_PROGRAM

// Application/UserCode/Sevcon_PSP/Sevcon_Steer_TxConversion_1
PROGRAM Sevcon_Steer_TxConversion_1
VAR
END_VAR
VAR CONSTANT
	SEVCON_TX_CF	:	REAL	:=	0.0625;
END_VAR




gu16_Sevcon1_TorqueRq_Tx				:=	REAL_TO_UINT(gr_Sevcon1_TorqueRq / SEVCON_TX_CF);
gu16_Sevcon1_TorqueTractionLimit_Tx		:=	REAL_TO_UINT(gr_Sevcon1_TorqueTractionLimit / SEVCON_TX_CF);
gu16_Sevcon1_TorqueRegenLimit_Tx		:=	REAL_TO_UINT(gr_Sevcon1_TorqueRegenLimit / SEVCON_TX_CF);
gu16_Sevcon1_DCLink_VoltageTarget_Tx	:=	REAL_TO_UINT(gr_Sevcon1_DCLink_VoltageTarget / SEVCON_TX_CF);
gu16_Sevcon1_DebugIqDirectControl_Tx	:=	REAL_TO_UINT(gr_Sevcon1_DebugIqDirectControl / SEVCON_TX_CF);
gu16_Sevcon1_DebugIdDirectControl_Tx	:=	REAL_TO_UINT(gr_Sevcon1_DebugIdDirectControl / SEVCON_TX_CF);

END_PROGRAM

// Application/UserCode/BMS/CATL/CATLBMS_RxConversion
PROGRAM CATLBMS_RxConversion

(*Convert input variables into real units by applying conversion factors and offsets*)

END_PROGRAM

// Application/UserCode/BMS/CATL/CATLBMS1_Rx_1
PROGRAM CATLBMS1_Rx_1

(*Program to receive all data from the CATL BMS*)



(*Initial saving CAN messages to receipt strucutres*)


(*Unpacking structures into variables*)


(*Comms loss check to ensure all messages are still being received*)


CATLBMS_RxConversion();

END_PROGRAM

// Application/UserCode/BMS/CATL/CATLBMS_RxConversion_1
PROGRAM CATLBMS_RxConversion_1

(*Convert input variables into real units by applying conversion factors and offsets*)

END_PROGRAM

// Application/UserCode/BMS/OrionBMS/Orion_Control_1
PROGRAM Orion_Control_1
VAR
	OrionPause_Timer	:	TON;
	hton_DisconnectionPause_Timer	:	TON;
END_VAR

(*Program to control the BMS during operation*)
(*Setting battery mode*)
IF (gu8_SystemState = DRIVE_SYS) THEN
	(*Have an initial short pause after contactors have closed before changing into discharge mode*)
	OrionPause_Timer(IN := TRUE, PT := T#20mS);
	IF (OrionPause_Timer.Q = TRUE) THEN
		(*Set discharge output*)
		DO_q_DrivetrainKL15C_DO	:=	FALSE;
		DO_q_DrivetrainKL15D_DO	:=	TRUE;
		(*Request on CAN the BMS into operational mode*)
		gu8_BMS1_MPO_1_State	:=	1;
		gu8_BMS1_MPO_2_State	:=	1; (* This does F_ALL *)
		gu8_BMS2_MPO_1_State	:=	1;
		gu8_BMS2_MPO_2_State	:=	1;
		
		
	END_IF
	hton_DisconnectionPause_Timer(IN := FALSE, PT := T#0MS);
ELSIF (gu8_SystemState = PLUGIN_SYS) THEN
	(*Have an initial short pause after contactors have closed before changing into charge mode*)
	OrionPause_Timer(IN := TRUE, PT := T#20MS);
	IF (OrionPause_Timer.Q = TRUE) THEN
		(*Set outputs for charge mode*)
		DO_q_DrivetrainKL15C_DO	:=	TRUE;
		DO_q_DrivetrainKL15D_DO	:=	FALSE;
		(*Request on CAN the BMS into operational mode*)
		gu8_BMS1_MPO_1_State	:=	0;
		gu8_BMS1_MPO_2_State	:=	0;
		gu8_BMS2_MPO_1_State	:=	0;
		gu8_BMS2_MPO_2_State	:=	0;
	END_IF
	hton_DisconnectionPause_Timer(IN := FALSE, PT := T#0MS);
ELSIF (DO_q_BatteryDischargeMain_DO = FALSE AND DO_q_Battery1ChargeMain_DO = FALSE AND DO_q_Battery2ChargeMain_DO = FALSE AND
		DO_q_BatteryDischargePrecharge_DO = FALSE AND DO_q_Battery1ChargePrecharge_DO = FALSE AND DO_q_Battery2ChargePrecharge_DO = FALSE) THEN
	(*Only perform disconnect of batteries when all contactors are opened to prevent them from damaging their own contactors Explain ??MAT *)
	hton_DisconnectionPause_Timer(IN := TRUE, PT := T#100MS);
	IF (hton_DisconnectionPause_Timer.Q = TRUE) THEN
		DO_q_DrivetrainKL15C_DO	:=	FALSE;
		DO_q_DrivetrainKL15D_DO	:=	FALSE;
		(*Request the BMS inactive*)
		gu8_BMS1_MPO_1_State	:=	0;
		gu8_BMS1_MPO_2_State	:=	0;
		gu8_BMS2_MPO_1_State	:=	0;
		gu8_BMS2_MPO_2_State	:=	0;
			
	END_IF
	OrionPause_Timer(IN := FALSE, PT := t#0ms);
END_IF
IF HMI_Rx.PB_BMS1_DTC_Reset THEN
	gu8_BMS1_MPO_3_State :=1;
	ELSE gu8_BMS1_MPO_3_State :=0;
END_IF
IF HMI_Rx.PB_BMS2_DTC_Reset THEN
	gu8_BMS2_MPO_3_State :=1;
	ELSE gu8_BMS2_MPO_3_State :=0;
END_IF

END_PROGRAM

// Application/UserCode/BMS/OrionBMS/OrionBMS1_Rx_1
PROGRAM OrionBMS1_Rx_1
VAR
	OrionBMS1_6B0_Rx	:	Receive_CAN2_STD;
	OrionBMS1_6B1_Rx	:	Receive_CAN2_STD;
	OrionBMS1_6B2_Rx	:	Receive_CAN2_STD;
	OrionBMS1_6B3_Rx	:	Receive_CAN2_STD;
	OrionBMS1_6B4_Rx	:	Receive_CAN2_STD;
	OrionBMS1_6B5_Rx	:	Receive_CAN2_STD;
	OrionBMS1_6B6_Rx	:	Receive_CAN2_STD;
	OrionBMS1_6B7_Rx	:	Receive_CAN2_STD;
	OrionBMS1_6B8_Rx	:	Receive_CAN2_STD;
	OrionBMS1_6B9_Rx	:	Receive_CAN2_STD;
	OrionBMS1_6BA_Rx	:	Receive_CAN2_STD;
	OrionBMS1_6BB_Rx	:	Receive_CAN2_STD;
	OrionBMS1_6BC_Rx	:	Receive_CAN2_STD;
	OrionBMS1_6BD_Rx	:	Receive_CAN2_STD;
	
	OrionBMS1_6B0_Rx_Timer	:	TON;
	OrionBMS1_6B1_Rx_Timer	:	TON;
	OrionBMS1_6B2_Rx_Timer	:	TON;
	OrionBMS1_6B3_Rx_Timer	:	TON;
	OrionBMS1_6B4_Rx_Timer	:	TON;
	OrionBMS1_6B5_Rx_Timer	:	TON;
	OrionBMS1_6B6_Rx_Timer	:	TON;
	OrionBMS1_6B7_Rx_Timer	:	TON;
	OrionBMS1_6B8_Rx_Timer	:	TON;
	OrionBMS1_6B9_Rx_Timer	:	TON;
	OrionBMS1_6BA_Rx_Timer	:	TON;
	OrionBMS1_6BB_Rx_Timer	:	TON;
	OrionBMS1_6BC_Rx_Timer	:	TON;
	OrionBMS1_6BD_Rx_Timer	:	TON;
	END_VAR

(*Program to receive all data from the Orion BMS*)
(*Initial saving CAN messages to receipt strucutres*)
OrionBMS1_6B0_Rx(u32_COBID	:=	16#6B0,
				 q_NewData => ,
				 au8_Data => ,
				 u8_Length => 			);
				 
OrionBMS1_6B1_Rx(u32_COBID	:=	16#6B1,
				 q_NewData => ,
				 au8_Data => ,
				 u8_Length => 			);
				 
OrionBMS1_6B2_Rx(u32_COBID	:=	16#6B2,
				 q_NewData => ,
				 au8_Data => ,
				 u8_Length => 			);
				 
OrionBMS1_6B3_Rx(u32_COBID	:=	16#6B3,
				 q_NewData => ,
				 au8_Data => ,
				 u8_Length => 			);
				 
OrionBMS1_6B4_Rx(u32_COBID	:=	16#6B4,
				 q_NewData => ,
				 au8_Data => ,
				 u8_Length => 			);
				 
OrionBMS1_6B5_Rx(u32_COBID	:=	16#6B5,
				 q_NewData => ,
				 au8_Data => ,
				 u8_Length => 			);
				 
OrionBMS1_6B6_Rx(u32_COBID	:=	16#6B6,
				 q_NewData => ,
				 au8_Data => ,
				 u8_Length => 			);
				 
OrionBMS1_6B7_Rx(u32_COBID	:=	16#6B7,
				 q_NewData => ,
				 au8_Data => ,
				 u8_Length => 			);
			 
OrionBMS1_6B8_Rx(u32_COBID	:=	16#6B8,
				 q_NewData => ,
				 au8_Data => ,
				 u8_Length => 			);
				 
OrionBMS1_6B9_Rx(u32_COBID	:=	16#6B9,
				 q_NewData => ,
				 au8_Data => ,
				 u8_Length => 			);
				 
OrionBMS1_6BA_Rx(u32_COBID	:=	16#6BA,
				 q_NewData => ,
				 au8_Data => ,
				 u8_Length => 			);
				 
OrionBMS1_6BB_Rx(u32_COBID	:=	16#6BB,
				 q_NewData => ,
				 au8_Data => ,
				 u8_Length => 			);
				 
OrionBMS1_6BC_Rx(u32_COBID	:=	16#6BC,
				 q_NewData => ,
				 au8_Data => ,
				 u8_Length => 			);
				 
OrionBMS1_6BD_Rx(u32_COBID	:=	16#6BD,
				 q_NewData => ,
				 au8_Data => ,
				 u8_Length => 			);


(*Unpacking structures into variables*)
(*6B0*)
gs16_OrionBMS1_PackCurrent	:=	USINT_TO_INT(OrionBMS1_6B0_Rx.au8_Data[0]) +
								SHL(USINT_TO_INT(OrionBMS1_6B0_Rx.au8_Data[1]), 8);
gu16_OrionBMS1_RAW_Pack_Voltage	:=	USINT_TO_UINT(OrionBMS1_6B0_Rx.au8_Data[2]) +
								SHL(USINT_TO_UINT(OrionBMS1_6B0_Rx.au8_Data[3]), 8);
gu8_OrionBMS1_RAW_SOC	:=	OrionBMS1_6B0_Rx.au8_Data[4];
gu16_OrionBMS1_RelayState	:=	USINT_TO_UINT(OrionBMS1_6B0_Rx.au8_Data[5]) +
								SHL(USINT_TO_UINT(OrionBMS1_6B0_Rx.au8_Data[6]), 8);
gu8_OrionBMS1_Custom_Flag_1	:=	OrionBMS1_6B0_Rx.au8_Data[7];

(*6B1*)
gu8_OrionBMS1_Isolation_ADC			:=	USINT_TO_UINT(OrionBMS1_6B1_Rx.au8_Data[0]) +
									SHL(USINT_TO_UINT(OrionBMS1_6B1_Rx.au8_Data[1]), 8);
gu8_OrionBMS1_Shortest_Wave			:=	USINT_TO_UINT(OrionBMS1_6B1_Rx.au8_Data[2]) +
									SHL(USINT_TO_UINT(OrionBMS1_6B1_Rx.au8_Data[3]), 8);
gu16_OrionBMS1_Isolation_Clipping	:=	USINT_TO_UINT(OrionBMS1_6B1_Rx.au8_Data[4]) +
									SHL(USINT_TO_UINT(OrionBMS1_6B1_Rx.au8_Data[5]), 8);
gu16_OrionBMS1_Isolation_Threshold	:=	USINT_TO_UINT(OrionBMS1_6B1_Rx.au8_Data[6]) +
									SHL(USINT_TO_UINT(OrionBMS1_6B1_Rx.au8_Data[7]), 8);
									
(*6B2*)
gu16_OrionBMS1_DTC_Flags1		:=	USINT_TO_UINT(OrionBMS1_6B2_Rx.au8_Data[0]) +
								SHL(USINT_TO_UINT(OrionBMS1_6B2_Rx.au8_Data[1]), 8);
gu16_OrionBMS1_DTC_Flags2		:=	USINT_TO_UINT(OrionBMS1_6B2_Rx.au8_Data[2]) +
								SHL(USINT_TO_UINT(OrionBMS1_6B2_Rx.au8_Data[3]), 8);
gu16_OrionBMS1_FailsafeStatus	:=	USINT_TO_UINT(OrionBMS1_6B2_Rx.au8_Data[4]) +
								SHL(USINT_TO_UINT(OrionBMS1_6B2_Rx.au8_Data[5]), 8);
gu16_OrionBMS1_Current_Limit_Status		:=	USINT_TO_UINT(OrionBMS1_6B2_Rx.au8_Data[6]) +
								SHL(USINT_TO_UINT(OrionBMS1_6B2_Rx.au8_Data[7]), 8);
(*6B3*)
gu8_OrionBMS1_PackHealth			:=	OrionBMS1_6B3_Rx.au8_Data[0];
gu16_OrionBMS1_PackCycles			:=	USINT_TO_UINT(OrionBMS1_6B3_Rx.au8_Data[1]) +
									SHL(USINT_TO_UINT(OrionBMS1_6B3_Rx.au8_Data[2]), 8);
gu16_OrionBMS1_PackResistance		:=	USINT_TO_UINT(OrionBMS1_6B3_Rx.au8_Data[3]) +
									SHL(USINT_TO_UINT(OrionBMS1_6B3_Rx.au8_Data[4]), 8);
gu8_OrionBMS1_PopulatedCells		:=	OrionBMS1_6B3_Rx.au8_Data[5];
gu16_OrionBMS1_MaximumPackVoltage	:=	USINT_TO_UINT (OrionBMS1_6B3_Rx.au8_Data[6]) +
									SHL(USINT_TO_UINT(OrionBMS1_6B3_Rx.au8_Data[7]),8);

(*6B4*)
gu8_OrionBMS1_HighTemp		:=	OrionBMS1_6B4_Rx.au8_Data[0];
gu8_OrionBMS1_LowTemp		:=	OrionBMS1_6B4_Rx.au8_Data[1];
gu8_OrionBMS1_AverageTemp	:=	OrionBMS1_6B4_Rx.au8_Data[2];
gu8_OrionBMS1_InternalTemp	:=	OrionBMS1_6B4_Rx.au8_Data[3];
gu16_OrionBMS1_MinimumPackVoltage	:=	USINT_TO_UINT(OrionBMS1_6B4_Rx.au8_Data[4]) +
									SHL(USINT_TO_UINT(OrionBMS1_6B4_Rx.au8_Data[5]), 8);
gu16_OrionBMS1_PackAmphours	:=	USINT_TO_UINT(OrionBMS1_6B4_Rx.au8_Data[6]) +
								SHL(USINT_TO_UINT(OrionBMS1_6B4_Rx.au8_Data[7]), 8);
(*6B5*)
gu16_OrionBMS1_AverageCellVoltage	:=	USINT_TO_UINT(OrionBMS1_6B5_Rx.au8_Data[0]) +
										SHL(USINT_TO_UINT(OrionBMS1_6B5_Rx.au8_Data[1]), 8);
gu16_OrionBMS1_LowCellVoltage		:=	USINT_TO_UINT(OrionBMS1_6B5_Rx.au8_Data[2]) +
										SHL(USINT_TO_UINT(OrionBMS1_6B5_Rx.au8_Data[3]), 8);
gu16_OrionBMS1_HighCellVoltage		:=	USINT_TO_UINT(OrionBMS1_6B5_Rx.au8_Data[4]) +
										SHL(USINT_TO_UINT(OrionBMS1_6B5_Rx.au8_Data[5]), 8);
gu8_OrionBMS1_LowCellVoltNumber		:=	OrionBMS1_6B5_Rx.au8_Data[6];
gu8_OrionBMS1_HighCellVoltNumber	:=	OrionBMS1_6B5_Rx.au8_Data[7];
(*6B6*)
gu8_OrionBMS1_Low_Intres_ID			:=	OrionBMS1_6B6_Rx.au8_Data[0];
gu8_OrionBMS1_High_Intres_ID		:=	OrionBMS1_6B6_Rx.au8_Data[1];
gu16_OrionBMS1_Low_Cell_Resistance	:=	USINT_TO_UINT(OrionBMS1_6B6_Rx.au8_Data[2]) +
										SHL(USINT_TO_UINT(OrionBMS1_6B6_Rx.au8_Data[3]), 8);
gu16_OrionBMS1_High_Cell_Resistance	:=	USINT_TO_UINT(OrionBMS1_6B6_Rx.au8_Data[4]) +
										SHL(USINT_TO_UINT(OrionBMS1_6B6_Rx.au8_Data[5]), 8);
gu16_OrionBMS1_Average_Cell_Resistance	:=	USINT_TO_UINT(OrionBMS1_6B6_Rx.au8_Data[6]) +
										SHL(USINT_TO_UINT(OrionBMS1_6B6_Rx.au8_Data[7]), 8);

(*6B7*)
gu8_OrionBMS1_Low_Thermistor_ID			:=	OrionBMS1_6B7_Rx.au8_Data[0];
gu8_OrionBMS1_High_Thermistor_ID		:=	OrionBMS1_6B7_Rx.au8_Data[1];
gu16_OrionBMS1_PackDCL				:=	USINT_TO_UINT(OrionBMS1_6B7_Rx.au8_Data[2]) +
										SHL(USINT_TO_UINT(OrionBMS1_6B7_Rx.au8_Data[3]), 8);
gu16_OrionBMS1_PackCCL				:=	USINT_TO_UINT(OrionBMS1_6B7_Rx.au8_Data[4]) +
										SHL(USINT_TO_UINT(OrionBMS1_6B7_Rx.au8_Data[5]), 8);
gu16_OrionBMS1_PackSummedVoltage	:=	USINT_TO_UINT(OrionBMS1_6B7_Rx.au8_Data[6]) +
										SHL(USINT_TO_UINT(OrionBMS1_6B7_Rx.au8_Data[7]), 8);

(*6B8*)
	gu8_OrionBMS1_Firmware_Minor		:=	OrionBMS1_6B8_Rx.au8_Data[0];	
	gu8_OrionBMS1_Firmware_Patch		:=	OrionBMS1_6B8_Rx.au8_Data[1];		
	gu8_OrionBMS1_Constant_2			:=	OrionBMS1_6B8_Rx.au8_Data[2];		
	gu8_OrionBMS1_Constant_3			:=	OrionBMS1_6B8_Rx.au8_Data[3];		
	gu8_OrionBMS1_Constant_4			:=	OrionBMS1_6B8_Rx.au8_Data[4];		
	gu16_OrionBMS1_CheckSum	:=	USINT_TO_UINT(OrionBMS1_6B8_Rx.au8_Data[5]) +
										SHL(USINT_TO_UINT(OrionBMS1_6B8_Rx.au8_Data[6]), 8);
	gu8_OrionBMS1_Spare_6B6_7			:=	OrionBMS1_6B8_Rx.au8_Data[7];


(*6B9*)
gu8_OrionBMS1_6B9_0		:=	OrionBMS1_6B9_Rx.au8_Data[0];
gu8_OrionBMS1_6B9_1		:=	OrionBMS1_6B9_Rx.au8_Data[1];
gu8_OrionBMS1_6B9_2		:=	OrionBMS1_6B9_Rx.au8_Data[2];
gu8_OrionBMS1_6B9_3		:=	OrionBMS1_6B9_Rx.au8_Data[3];
gu8_OrionBMS1_6B9_4		:=	OrionBMS1_6B9_Rx.au8_Data[4];
gu8_OrionBMS1_6B9_5		:=	OrionBMS1_6B9_Rx.au8_Data[5];
gu8_OrionBMS1_6B9_6		:=	OrionBMS1_6B9_Rx.au8_Data[6];
gu8_OrionBMS1_6B9_7		:=	OrionBMS1_6B9_Rx.au8_Data[7];


(*6BA*)
gu8_OrionBMS1_6BA_0		:=	OrionBMS1_6BA_Rx.au8_Data[0];
gu8_OrionBMS1_6BA_1		:=	OrionBMS1_6BA_Rx.au8_Data[1];
gu8_OrionBMS1_6BA_2		:=	OrionBMS1_6BA_Rx.au8_Data[2];
gu8_OrionBMS1_6BA_3		:=	OrionBMS1_6BA_Rx.au8_Data[3];
gu8_OrionBMS1_6BA_4		:=	OrionBMS1_6BA_Rx.au8_Data[4];
gu8_OrionBMS1_6BA_5		:=	OrionBMS1_6BA_Rx.au8_Data[5];
gu8_OrionBMS1_6BA_6		:=	OrionBMS1_6BA_Rx.au8_Data[6];
gu8_OrionBMS1_6BA_7		:=	OrionBMS1_6BA_Rx.au8_Data[7];

(*6BB*)
gu8_OrionBMS1_6BB_0		:=	OrionBMS1_6BB_Rx.au8_Data[0];
gu8_OrionBMS1_6BB_1		:=	OrionBMS1_6BB_Rx.au8_Data[1];
gu8_OrionBMS1_6BB_2		:=	OrionBMS1_6BB_Rx.au8_Data[2];
gu8_OrionBMS1_6BB_3		:=	OrionBMS1_6BB_Rx.au8_Data[3];
gu8_OrionBMS1_6BB_4		:=	OrionBMS1_6BB_Rx.au8_Data[4];
gu8_OrionBMS1_6BB_5		:=	OrionBMS1_6BB_Rx.au8_Data[5];
gu8_OrionBMS1_6BB_6		:=	OrionBMS1_6BB_Rx.au8_Data[6];
gu8_OrionBMS1_6BB_7		:=	OrionBMS1_6BB_Rx.au8_Data[7];

(*6BC*)
gu8_OrionBMS1_6BC_0		:=	OrionBMS1_6BC_Rx.au8_Data[0];
gu8_OrionBMS1_6BC_1		:=	OrionBMS1_6BC_Rx.au8_Data[1];
gu8_OrionBMS1_6BC_2		:=	OrionBMS1_6BC_Rx.au8_Data[2];
gu8_OrionBMS1_6BC_3		:=	OrionBMS1_6BC_Rx.au8_Data[3];
gu8_OrionBMS1_6BC_4		:=	OrionBMS1_6BC_Rx.au8_Data[4];
gu8_OrionBMS1_6BC_5		:=	OrionBMS1_6BC_Rx.au8_Data[5];
gu8_OrionBMS1_6BC_6		:=	OrionBMS1_6BC_Rx.au8_Data[6];
gu8_OrionBMS1_6BC_7		:=	OrionBMS1_6BC_Rx.au8_Data[7];	
	
(*6BD*)
gu8_OrionBMS1_6BD_0		:=	OrionBMS1_6BD_Rx.au8_Data[0];
gu8_OrionBMS1_6BD_1		:=	OrionBMS1_6BD_Rx.au8_Data[1];
gu8_OrionBMS1_6BD_2		:=	OrionBMS1_6BD_Rx.au8_Data[2];
gu8_OrionBMS1_6BD_3		:=	OrionBMS1_6BD_Rx.au8_Data[3];
gu8_OrionBMS1_6BD_4		:=	OrionBMS1_6BD_Rx.au8_Data[4];
gu8_OrionBMS1_6BD_5		:=	OrionBMS1_6BD_Rx.au8_Data[5];
gu8_OrionBMS1_6BD_6		:=	OrionBMS1_6BD_Rx.au8_Data[6];
gu8_OrionBMS1_6BD_7		:=	OrionBMS1_6BD_Rx.au8_Data[7];

(*Comms loss check to ensure all messages are still being received*)
OrionBMS1_6B0_Rx_Timer(IN := NOT(OrionBMS1_6B0_Rx.q_NewData), PT := T#3S);
OrionBMS1_6B1_Rx_Timer(IN := NOT(OrionBMS1_6B1_Rx.q_NewData), PT := T#3S);
OrionBMS1_6B2_Rx_Timer(IN := NOT(OrionBMS1_6B2_Rx.q_NewData), PT := T#3S);
OrionBMS1_6B3_Rx_Timer(IN := NOT(OrionBMS1_6B3_Rx.q_NewData), PT := T#3S);
OrionBMS1_6B4_Rx_Timer(IN := NOT(OrionBMS1_6B4_Rx.q_NewData), PT := T#3S);
OrionBMS1_6B5_Rx_Timer(IN := NOT(OrionBMS1_6B5_Rx.q_NewData), PT := T#3S);
OrionBMS1_6B6_Rx_Timer(IN := NOT(OrionBMS1_6B6_Rx.q_NewData), PT := T#3S);
OrionBMS1_6B7_Rx_Timer(IN := NOT(OrionBMS1_6B7_Rx.q_NewData), PT := T#3S);
OrionBMS1_6B8_Rx_Timer(IN := NOT(OrionBMS1_6B8_Rx.q_NewData), PT := T#3S);
OrionBMS1_6B9_Rx_Timer(IN := NOT(OrionBMS1_6B9_Rx.q_NewData), PT := T#3S);
OrionBMS1_6BA_Rx_Timer(IN := NOT(OrionBMS1_6BA_Rx.q_NewData), PT := T#3S);
OrionBMS1_6BB_Rx_Timer(IN := NOT(OrionBMS1_6BB_Rx.q_NewData), PT := T#3S);
OrionBMS1_6BC_Rx_Timer(IN := NOT(OrionBMS1_6BC_Rx.q_NewData), PT := T#3S);
OrionBMS1_6BD_Rx_Timer(IN := NOT(OrionBMS1_6BD_Rx.q_NewData), PT := T#3S);
IF (OrionBMS1_6B0_Rx_Timer.Q = TRUE AND OrionBMS1_6B1_Rx_Timer.Q = TRUE AND OrionBMS1_6B2_Rx_Timer.Q = TRUE AND
	OrionBMS1_6B3_Rx_Timer.Q = TRUE AND OrionBMS1_6B4_Rx_Timer.Q = TRUE AND OrionBMS1_6B5_Rx_Timer.Q = TRUE AND
	OrionBMS1_6B6_Rx_Timer.Q = TRUE AND OrionBMS1_6B7_Rx_Timer.Q = TRUE AND OrionBMS1_6B8_Rx_Timer.Q = TRUE AND
	OrionBMS1_6B9_Rx_Timer.Q = TRUE AND OrionBMS1_6BA_Rx_Timer.Q = TRUE AND OrionBMS1_6BB_Rx_Timer.Q = TRUE AND
	OrionBMS1_6BC_Rx_Timer.Q = TRUE AND OrionBMS1_6BD_Rx_Timer.Q = TRUE											) THEN

	gq_OrionBMS1_CommsLoss	:=	TRUE;
ELSE
	gq_OrionBMS1_CommsLoss	:=	FALSE;
END_IF


OrionBMS1_RxConversion();

END_PROGRAM

// Application/UserCode/BMS/OrionBMS/OrionBMS1_RxConversion_1
PROGRAM OrionBMS1_RxConversion_1
VAR
	gr_OrionBMS1_PackVoltage			:REAL;
	gr_OrionBMS1_PackCurrent			:REAL;
	gr_OrionBMS1_PackSOC				:REAL;
	gr_OrionBMS1_Max_Charging_Voltage	:REAL;
	gq_BMS1_BalActive					:BOOL;
	gq_BMS1_Flag_1						:BOOL;
	gq_BMS1_Flag_2						:BOOL;
	gq_BMS1_Flag_3						:BOOL;
	gq_BMS1_Flag_4						:BOOL;
	gq_BMS1_Flag_5						:BOOL;
	gq_BMS1_Flag_6						:BOOL;
	Safety_OK   : BOOL;
END_VAR
VAR CONSTANT
	SYSTEMRX_CF	:	REAL	:=	0.1;
	CURRENT_CF	:	REAL	:=	0.1;
END_VAR

(*Convert input variables into real units by applying conversion factors and offsets*)

gr_OrionBMS1_PackVoltage			:=	UINT_TO_REAL(gu16_OrionBMS1_RAW_Pack_Voltage) * SYSTEMRX_CF;
gr_OrionBMS1_PackCurrent			:=	INT_TO_REAL(gs16_OrionBMS1_PackCurrent) * CURRENT_CF;
gr_OrionBMS1_PackSOC				:=	REAL_TO_USINT(gu8_OrionBMS1_RAW_SOC / 2);
gr_OrionBMS1_Max_Charging_Voltage	:= gu8_OrionBMS1_PopulatedCells *3.65;

OrionBMS1_DTCFlag1_0A07_DischargeLimitEnforcementFault		:=	gu16_OrionBMS1_DTC_Flags1.0;
OrionBMS1_DTCFlag1_0A08_ChargerSafetyRelayFault 			:=	gu16_OrionBMS1_DTC_Flags1.1;
OrionBMS1_DTCFlag1_0A09_InternalHardwareFault				:=	gu16_OrionBMS1_DTC_Flags1.2;
OrionBMS1_DTCFlag1_0A0A_InternalHeatskinkThermistorFault 	:=	gu16_OrionBMS1_DTC_Flags1.3;
OrionBMS1_DTCFlag1_0A0B_InternalSoftwareFault				:=	gu16_OrionBMS1_DTC_Flags1.4;
OrionBMS1_DTCFlag1_0A0C_HighestCellVoltageTooHighFault 	:=	gu16_OrionBMS1_DTC_Flags1.5;
OrionBMS1_DTCFlag1_0A0E_LowestCellVoltageTooLowFault 		:=	gu16_OrionBMS1_DTC_Flags1.6;
OrionBMS1_DTCFlag1_0A10_PackTooHotFault 					:=	gu16_OrionBMS1_DTC_Flags1.7;
OrionBMS1_DTCFlags_Reserved_Bit8 							:=	gu16_OrionBMS1_DTC_Flags1.8;
OrionBMS1_DTCFlags_Reserved_Bit9 							:=	gu16_OrionBMS1_DTC_Flags1.9;
OrionBMS1_DTCFlags_Reserved_Bit10 							:=	gu16_OrionBMS1_DTC_Flags1.10;
OrionBMS1_DTCFlags_Reserved_Bit11 							:=	gu16_OrionBMS1_DTC_Flags1.11;
OrionBMS1_DTCFlags_Reserved_Bit12 							:=	gu16_OrionBMS1_DTC_Flags1.12;
OrionBMS1_DTCFlags_Reserved_Bit13 							:=	gu16_OrionBMS1_DTC_Flags1.13;
OrionBMS1_DTCFlags_Reserved_Bit14 							:=	gu16_OrionBMS1_DTC_Flags1.14;
OrionBMS1_DTCFlags_Reserved_Bit15							:=	gu16_OrionBMS1_DTC_Flags1.15;

OrionBMS1_DTCFlags2_0A1F_InternalCommunicationFault			:=	gu16_OrionBMS1_DTC_Flags2.0;
OrionBMS1_DTCFlags2_0A12_CellBalancingStruckOffFault		:=	gu16_OrionBMS1_DTC_Flags2.1;
OrionBMS1_DTCFlags2_0A80_WeakCellFault						:=	gu16_OrionBMS1_DTC_Flags2.2;
OrionBMS1_DTCFlags2_0AFA_LowCellVoltageFault				:=	gu16_OrionBMS1_DTC_Flags2.3;
OrionBMS1_DTCFlags2_0A04_OpenWiringFault					:=	gu16_OrionBMS1_DTC_Flags2.4;
OrionBMS1_DTCFlags2_0AC0_CurrentSensorFault					:=	gu16_OrionBMS1_DTC_Flags2.5;
OrionBMS1_DTCFlags2_0A0D_HighestCellVoltageOver5vFault		:=	gu16_OrionBMS1_DTC_Flags2.6;
OrionBMS1_DTCFlags2_0A0F_CellASICFault						:=	gu16_OrionBMS1_DTC_Flags2.7;
OrionBMS1_DTCFlags2_0A02_WeakPackFault						:=	gu16_OrionBMS1_DTC_Flags2.8;
OrionBMS1_DTCFlags2_0A81_FanMonitorFault					:=	gu16_OrionBMS1_DTC_Flags2.9;
OrionBMS1_DTCFlags2_0A9C_ThermistorFault					:=	gu16_OrionBMS1_DTC_Flags2.10;
OrionBMS1_DTCFlags2_0100_ExternalCommunicationFault			:=	gu16_OrionBMS1_DTC_Flags2.11;
OrionBMS1_DTCFlags2_0560_RedundantPowerSupplyFault			:=	gu16_OrionBMS1_DTC_Flags2.12;
OrionBMS1_DTCFlags2_0AA6_HighVoltageIsolatonFault			:=	gu16_OrionBMS1_DTC_Flags2.13;
OrionBMS1_DTCFlags2_0A05_InputPowerSupplyFault				:=	gu16_OrionBMS1_DTC_Flags2.14;
OrionBMS1_DTCFlags2_0A06_ChargeLimitEnforcementFault		:=	gu16_OrionBMS1_DTC_Flags2.15;

gq_BMS1_BalActive			:=	gu8_OrionBMS1_Custom_Flag_1.0;
gq_BMS1_Flag_1				:=	gu8_OrionBMS1_Custom_Flag_1.1;
gq_BMS1_Flag_2				:=	gu8_OrionBMS1_Custom_Flag_1.2;
gq_BMS1_Flag_3				:=	gu8_OrionBMS1_Custom_Flag_1.3;
gq_BMS1_Flag_4				:=	gu8_OrionBMS1_Custom_Flag_1.4;
gq_BMS1_Flag_5				:=	gu8_OrionBMS1_Custom_Flag_1.5;
gq_BMS1_Flag_6				:=	gu8_OrionBMS1_Custom_Flag_1.6;
Safety_OK				:=	gu8_OrionBMS1_Custom_Flag_1.7;

END_PROGRAM

// Application/UserCode/BMS/OrionBMS/OrionBMS2_Rx_1
PROGRAM OrionBMS2_Rx_1
VAR
	OrionBMS2_6B0_Rx	:	Receive_CAN3_STD;
	OrionBMS2_6B1_Rx	:	Receive_CAN3_STD;
	OrionBMS2_6B2_Rx	:	Receive_CAN3_STD;
	OrionBMS2_6B3_Rx	:	Receive_CAN3_STD;
	OrionBMS2_6B4_Rx	:	Receive_CAN3_STD;
	OrionBMS2_6B5_Rx	:	Receive_CAN3_STD;
	OrionBMS2_6B6_Rx	:	Receive_CAN3_STD;
	OrionBMS2_6B7_Rx	:	Receive_CAN3_STD;
	OrionBMS2_6B8_Rx	:	Receive_CAN3_STD;
	OrionBMS2_6B9_Rx	:	Receive_CAN3_STD;
	OrionBMS2_6BA_Rx	:	Receive_CAN3_STD;
	OrionBMS2_6BB_Rx	:	Receive_CAN3_STD;
	OrionBMS2_6BC_Rx	:	Receive_CAN3_STD;
	OrionBMS2_6BD_Rx	:	Receive_CAN3_STD;
	
	OrionBMS2_6B0_Rx_Timer	:	TON;
	OrionBMS2_6B1_Rx_Timer	:	TON;
	OrionBMS2_6B2_Rx_Timer	:	TON;
	OrionBMS2_6B3_Rx_Timer	:	TON;
	OrionBMS2_6B4_Rx_Timer	:	TON;
	OrionBMS2_6B5_Rx_Timer	:	TON;
	OrionBMS2_6B6_Rx_Timer	:	TON;
	OrionBMS2_6B7_Rx_Timer	:	TON;
	OrionBMS2_6B8_Rx_Timer	:	TON;
	OrionBMS2_6B9_Rx_Timer	:	TON;
	OrionBMS2_6BA_Rx_Timer	:	TON;
	OrionBMS2_6BB_Rx_Timer	:	TON;
	OrionBMS2_6BC_Rx_Timer	:	TON;
	OrionBMS2_6BD_Rx_Timer	:	TON;
	END_VAR

(*Program to receive all data from the Orion BMS*)
(*Initial saving CAN messages to receipt strucutres*)
OrionBMS2_6B0_Rx(u32_COBID	:=	16#6B0,
				 q_NewData => ,
				 au8_Data => ,
				 u8_Length => 			);
				 
OrionBMS2_6B1_Rx(u32_COBID	:=	16#6B1,
				 q_NewData => ,
				 au8_Data => ,
				 u8_Length => 			);
				 
OrionBMS2_6B2_Rx(u32_COBID	:=	16#6B2,
				 q_NewData => ,
				 au8_Data => ,
				 u8_Length => 			);
				 
OrionBMS2_6B3_Rx(u32_COBID	:=	16#6B3,
				 q_NewData => ,
				 au8_Data => ,
				 u8_Length => 			);
				 
OrionBMS2_6B4_Rx(u32_COBID	:=	16#6B4,
				 q_NewData => ,
				 au8_Data => ,
				 u8_Length => 			);
				 
OrionBMS2_6B5_Rx(u32_COBID	:=	16#6B5,
				 q_NewData => ,
				 au8_Data => ,
				 u8_Length => 			);
				 
OrionBMS2_6B6_Rx(u32_COBID	:=	16#6B6,
				 q_NewData => ,
				 au8_Data => ,
				 u8_Length => 			);
				 
OrionBMS2_6B7_Rx(u32_COBID	:=	16#6B7,
				 q_NewData => ,
				 au8_Data => ,
				 u8_Length => 			);
			 
OrionBMS2_6B8_Rx(u32_COBID	:=	16#6B8,
				 q_NewData => ,
				 au8_Data => ,
				 u8_Length => 			);
				 
OrionBMS2_6B9_Rx(u32_COBID	:=	16#6B9,
				 q_NewData => ,
				 au8_Data => ,
				 u8_Length => 			);
				 
OrionBMS2_6BA_Rx(u32_COBID	:=	16#6BA,
				 q_NewData => ,
				 au8_Data => ,
				 u8_Length => 			);
				 
OrionBMS2_6BB_Rx(u32_COBID	:=	16#6BB,
				 q_NewData => ,
				 au8_Data => ,
				 u8_Length => 			);
				 
OrionBMS2_6BC_Rx(u32_COBID	:=	16#6BC,
				 q_NewData => ,
				 au8_Data => ,
				 u8_Length => 			);
				 
OrionBMS2_6BD_Rx(u32_COBID	:=	16#6BD,
				 q_NewData => ,
				 au8_Data => ,
				 u8_Length => 			);


(*Unpacking input structures into variables*)
(*6B0*)

gs16_OrionBMS2_PackCurrent	:=	USINT_TO_INT(OrionBMS2_6B0_Rx.au8_Data[0]) +
								SHL(USINT_TO_INT(OrionBMS2_6B0_Rx.au8_Data[1]), 8);
gu16_OrionBMS2_PackVoltage	:=	USINT_TO_UINT(OrionBMS2_6B0_Rx.au8_Data[2]) +
								SHL(USINT_TO_UINT(OrionBMS2_6B0_Rx.au8_Data[3]), 8);
gu8_OrionBMS2_RAW_SOC	:=	OrionBMS2_6B0_Rx.au8_Data[4];
gu16_OrionBMS2_RelayState	:=	USINT_TO_UINT(OrionBMS2_6B0_Rx.au8_Data[5]) +
								SHL(USINT_TO_UINT(OrionBMS2_6B0_Rx.au8_Data[6]), 8);
gu8_OrionBMS2_Custom_Flag_1	:=	OrionBMS2_6B0_Rx.au8_Data[7];

(*6B1*)
gu8_OrionBMS2_Isolation_ADC			:=	USINT_TO_UINT(OrionBMS2_6B1_Rx.au8_Data[0]) +
									SHL(USINT_TO_UINT(OrionBMS2_6B1_Rx.au8_Data[1]), 8);
gu8_OrionBMS2_Shortest_Wave			:=	USINT_TO_UINT(OrionBMS2_6B1_Rx.au8_Data[2]) +
									SHL(USINT_TO_UINT(OrionBMS2_6B1_Rx.au8_Data[3]), 8);
gu16_OrionBMS2_Isolation_Clipping	:=	USINT_TO_UINT(OrionBMS2_6B1_Rx.au8_Data[4]) +
									SHL(USINT_TO_UINT(OrionBMS2_6B1_Rx.au8_Data[5]), 8);
gu16_OrionBMS2_Isolation_Threshold	:=	USINT_TO_UINT(OrionBMS2_6B1_Rx.au8_Data[6]) +
									SHL(USINT_TO_UINT(OrionBMS2_6B1_Rx.au8_Data[7]), 8);
									
(*6B2*)
gu16_OrionBMS2_DTC_Flags1		:=	USINT_TO_UINT(OrionBMS2_6B2_Rx.au8_Data[0]) +
								SHL(USINT_TO_UINT(OrionBMS2_6B2_Rx.au8_Data[1]), 8);
gu16_OrionBMS2_DTC_Flags2		:=	USINT_TO_UINT(OrionBMS2_6B2_Rx.au8_Data[2]) +
								SHL(USINT_TO_UINT(OrionBMS2_6B2_Rx.au8_Data[3]), 8);
gu16_OrionBMS2_FailsafeStatus	:=	USINT_TO_UINT(OrionBMS2_6B2_Rx.au8_Data[4]) +
								SHL(USINT_TO_UINT(OrionBMS2_6B2_Rx.au8_Data[5]), 8);
gu16_OrionBMS2_CurrentLimit		:=	USINT_TO_UINT(OrionBMS2_6B2_Rx.au8_Data[6]) +
								SHL(USINT_TO_UINT(OrionBMS2_6B2_Rx.au8_Data[7]), 8);
(*6B3*)
gu8_OrionBMS2_PackHealth			:=	OrionBMS2_6B3_Rx.au8_Data[0];
gu16_OrionBMS2_PackCycles			:=	USINT_TO_UINT(OrionBMS2_6B3_Rx.au8_Data[1]) +
									SHL(USINT_TO_UINT(OrionBMS2_6B3_Rx.au8_Data[2]), 8);
gu16_OrionBMS2_PackResistance		:=	USINT_TO_UINT(OrionBMS2_6B3_Rx.au8_Data[3]) +
									SHL(USINT_TO_UINT(OrionBMS2_6B3_Rx.au8_Data[4]), 8);
gu8_OrionBMS2_PopulatedCells		:=	OrionBMS2_6B3_Rx.au8_Data[5];
gu16_OrionBMS2_MaximumPackVoltage	:=	USINT_TO_UINT (OrionBMS2_6B3_Rx.au8_Data[6]) +
									SHL(USINT_TO_UINT(OrionBMS2_6B3_Rx.au8_Data[7]),8);

(*6B4*)
gu8_OrionBMS2_HighTemp		:=	OrionBMS2_6B4_Rx.au8_Data[0];
gu8_OrionBMS2_LowTemp		:=	OrionBMS2_6B4_Rx.au8_Data[1];
gu8_OrionBMS2_AverageTemp	:=	OrionBMS2_6B4_Rx.au8_Data[2];
gu8_OrionBMS2_InternalTemp	:=	OrionBMS2_6B4_Rx.au8_Data[3];
gu16_OrionBMS2_MinimumPackVoltage	:=	USINT_TO_UINT(OrionBMS2_6B4_Rx.au8_Data[4]) +
									SHL(USINT_TO_UINT(OrionBMS2_6B4_Rx.au8_Data[5]), 8);
gu16_OrionBMS2_PackAmphours	:=	USINT_TO_UINT(OrionBMS2_6B4_Rx.au8_Data[6]) +
								SHL(USINT_TO_UINT(OrionBMS2_6B4_Rx.au8_Data[7]), 8);
(*6B5*)
gu16_OrionBMS2_AverageCellVoltage	:=	USINT_TO_UINT(OrionBMS2_6B5_Rx.au8_Data[0]) +
										SHL(USINT_TO_UINT(OrionBMS2_6B5_Rx.au8_Data[1]), 8);
gu16_OrionBMS2_LowCellVoltage		:=	USINT_TO_UINT(OrionBMS2_6B5_Rx.au8_Data[2]) +
										SHL(USINT_TO_UINT(OrionBMS2_6B5_Rx.au8_Data[3]), 8);
gu16_OrionBMS2_HighCellVoltage		:=	USINT_TO_UINT(OrionBMS2_6B5_Rx.au8_Data[4]) +
										SHL(USINT_TO_UINT(OrionBMS2_6B5_Rx.au8_Data[5]), 8);
gu8_OrionBMS2_LowCellVoltNumber		:=	OrionBMS2_6B5_Rx.au8_Data[6];
gu8_OrionBMS2_HighCellVoltNumber	:=	OrionBMS2_6B5_Rx.au8_Data[7];
(*6B6*)
gu8_OrionBMS2_Low_Intres_ID			:=	OrionBMS2_6B6_Rx.au8_Data[0];
gu8_OrionBMS2_High_Intres_ID		:=	OrionBMS2_6B6_Rx.au8_Data[1];
gu16_OrionBMS2_Low_Cell_Resistance	:=	USINT_TO_UINT(OrionBMS2_6B6_Rx.au8_Data[2]) +
										SHL(USINT_TO_UINT(OrionBMS2_6B6_Rx.au8_Data[3]), 8);
gu16_OrionBMS2_High_Cell_Resistance	:=	USINT_TO_UINT(OrionBMS2_6B6_Rx.au8_Data[4]) +
										SHL(USINT_TO_UINT(OrionBMS2_6B6_Rx.au8_Data[5]), 8);
gu16_OrionBMS2_Average_Cell_Resistance	:=	USINT_TO_UINT(OrionBMS2_6B6_Rx.au8_Data[6]) +
										SHL(USINT_TO_UINT(OrionBMS2_6B6_Rx.au8_Data[7]), 8);

(*6B7*)
gu8_OrionBMS2_Low_Thermistor_ID			:=	OrionBMS2_6B7_Rx.au8_Data[0];
gu8_OrionBMS2_High_Thermistor_ID		:=	OrionBMS2_6B7_Rx.au8_Data[1];
gu16_OrionBMS2_PackDCL				:=	USINT_TO_UINT(OrionBMS2_6B7_Rx.au8_Data[2]) +
										SHL(USINT_TO_UINT(OrionBMS2_6B7_Rx.au8_Data[3]), 8);
gu16_OrionBMS2_PackCCL				:=	USINT_TO_UINT(OrionBMS2_6B7_Rx.au8_Data[4]) +
										SHL(USINT_TO_UINT(OrionBMS2_6B7_Rx.au8_Data[5]), 8);
gu16_OrionBMS2_PackSummedVoltage	:=	USINT_TO_UINT(OrionBMS2_6B7_Rx.au8_Data[6]) +
										SHL(USINT_TO_UINT(OrionBMS2_6B7_Rx.au8_Data[7]), 8);

(*6B8*)
	gu8_OrionBMS2_Firmware_Minor	:=	OrionBMS2_6B8_Rx.au8_Data[0];	
	gu8_OrionBMS2_Firmware_Patch	:=	OrionBMS2_6B8_Rx.au8_Data[1];		
	gu8_OrionBMS2_Constant_2		:=	OrionBMS2_6B8_Rx.au8_Data[2];		
	gu8_OrionBMS2_Constant_3		:=	OrionBMS2_6B8_Rx.au8_Data[3];		
	gu8_OrionBMS2_Constant_4		:=	OrionBMS2_6B8_Rx.au8_Data[4];		
	gu16_OrionBMS2_CheckSum			:=	USINT_TO_UINT(OrionBMS2_6B8_Rx.au8_Data[5]) +
										SHL(USINT_TO_UINT(OrionBMS2_6B8_Rx.au8_Data[6]), 8);
	gu8_OrionBMS2_Spare_6B6_7	:=	OrionBMS2_6B8_Rx.au8_Data[7];


(*6B9*)
gu8_OrionBMS2_6B9_0		:=	OrionBMS2_6B9_Rx.au8_Data[0];
gu8_OrionBMS2_6B9_1		:=	OrionBMS2_6B9_Rx.au8_Data[1];
gu8_OrionBMS2_6B9_2		:=	OrionBMS2_6B9_Rx.au8_Data[2];
gu8_OrionBMS2_6B9_3		:=	OrionBMS2_6B9_Rx.au8_Data[3];
gu8_OrionBMS2_6B9_4		:=	OrionBMS2_6B9_Rx.au8_Data[4];
gu8_OrionBMS2_6B9_5		:=	OrionBMS2_6B9_Rx.au8_Data[5];
gu8_OrionBMS2_6B9_6		:=	OrionBMS2_6B9_Rx.au8_Data[6];
gu8_OrionBMS2_6B9_7		:=	OrionBMS2_6B9_Rx.au8_Data[7];


(*6BA*)
gu8_OrionBMS2_6BA_0		:=	OrionBMS2_6BA_Rx.au8_Data[0];
gu8_OrionBMS2_6BA_1		:=	OrionBMS2_6BA_Rx.au8_Data[1];
gu8_OrionBMS2_6BA_2		:=	OrionBMS2_6BA_Rx.au8_Data[2];
gu8_OrionBMS2_6BA_3		:=	OrionBMS2_6BA_Rx.au8_Data[3];
gu8_OrionBMS2_6BA_4		:=	OrionBMS2_6BA_Rx.au8_Data[4];
gu8_OrionBMS2_6BA_5		:=	OrionBMS2_6BA_Rx.au8_Data[5];
gu8_OrionBMS2_6BA_6		:=	OrionBMS2_6BA_Rx.au8_Data[6];
gu8_OrionBMS2_6BA_7		:=	OrionBMS2_6BA_Rx.au8_Data[7];

(*6BB*)
gu8_OrionBMS2_6BB_0		:=	OrionBMS2_6BB_Rx.au8_Data[0];
gu8_OrionBMS2_6BB_1		:=	OrionBMS2_6BB_Rx.au8_Data[1];
gu8_OrionBMS2_6BB_2		:=	OrionBMS2_6BB_Rx.au8_Data[2];
gu8_OrionBMS2_6BB_3		:=	OrionBMS2_6BB_Rx.au8_Data[3];
gu8_OrionBMS2_6BB_4		:=	OrionBMS2_6BB_Rx.au8_Data[4];
gu8_OrionBMS2_6BB_5		:=	OrionBMS2_6BB_Rx.au8_Data[5];
gu8_OrionBMS2_6BB_6		:=	OrionBMS2_6BB_Rx.au8_Data[6];
gu8_OrionBMS2_6BB_7		:=	OrionBMS2_6BB_Rx.au8_Data[7];

(*6BC*)
gu8_OrionBMS2_6BC_0		:=	OrionBMS2_6BC_Rx.au8_Data[0];
gu8_OrionBMS2_6BC_1		:=	OrionBMS2_6BC_Rx.au8_Data[1];
gu8_OrionBMS2_6BC_2		:=	OrionBMS2_6BC_Rx.au8_Data[2];
gu8_OrionBMS2_6BC_3		:=	OrionBMS2_6BC_Rx.au8_Data[3];
gu8_OrionBMS2_6BC_4		:=	OrionBMS2_6BC_Rx.au8_Data[4];
gu8_OrionBMS2_6BC_5		:=	OrionBMS2_6BC_Rx.au8_Data[5];
gu8_OrionBMS2_6BC_6		:=	OrionBMS2_6BC_Rx.au8_Data[6];
gu8_OrionBMS2_6BC_7		:=	OrionBMS2_6BC_Rx.au8_Data[7];	
	
(*6BD*)
gu8_OrionBMS2_6BD_0		:=	OrionBMS2_6BD_Rx.au8_Data[0];
gu8_OrionBMS2_6BD_1		:=	OrionBMS2_6BD_Rx.au8_Data[1];
gu8_OrionBMS2_6BD_2		:=	OrionBMS2_6BD_Rx.au8_Data[2];
gu8_OrionBMS2_6BD_3		:=	OrionBMS2_6BD_Rx.au8_Data[3];
gu8_OrionBMS2_6BD_4		:=	OrionBMS2_6BD_Rx.au8_Data[4];
gu8_OrionBMS2_6BD_5		:=	OrionBMS2_6BD_Rx.au8_Data[5];
gu8_OrionBMS2_6BD_6		:=	OrionBMS2_6BD_Rx.au8_Data[6];
gu8_OrionBMS2_6BD_7		:=	OrionBMS2_6BD_Rx.au8_Data[7];


(*Communications loss check*)
OrionBMS2_6B0_Rx_Timer(IN := NOT(OrionBMS2_6B0_Rx.q_NewData), PT := T#3S);
OrionBMS2_6B1_Rx_Timer(IN := NOT(OrionBMS2_6B1_Rx.q_NewData), PT := T#3S);
OrionBMS2_6B2_Rx_Timer(IN := NOT(OrionBMS2_6B2_Rx.q_NewData), PT := T#3S);
OrionBMS2_6B3_Rx_Timer(IN := NOT(OrionBMS2_6B3_Rx.q_NewData), PT := T#3S);
OrionBMS2_6B4_Rx_Timer(IN := NOT(OrionBMS2_6B4_Rx.q_NewData), PT := T#3S);
OrionBMS2_6B5_Rx_Timer(IN := NOT(OrionBMS2_6B5_Rx.q_NewData), PT := T#3S);
OrionBMS2_6B6_Rx_Timer(IN := NOT(OrionBMS2_6B6_Rx.q_NewData), PT := T#3S);
OrionBMS2_6B7_Rx_Timer(IN := NOT(OrionBMS2_6B7_Rx.q_NewData), PT := T#3S);
OrionBMS2_6B8_Rx_Timer(IN := NOT(OrionBMS2_6B8_Rx.q_NewData), PT := T#3S);
OrionBMS2_6B9_Rx_Timer(IN := NOT(OrionBMS2_6B9_Rx.q_NewData), PT := T#3S);
OrionBMS2_6BA_Rx_Timer(IN := NOT(OrionBMS2_6BA_Rx.q_NewData), PT := T#3S);
OrionBMS2_6BB_Rx_Timer(IN := NOT(OrionBMS2_6BB_Rx.q_NewData), PT := T#3S);
OrionBMS2_6BC_Rx_Timer(IN := NOT(OrionBMS2_6BC_Rx.q_NewData), PT := T#3S);
OrionBMS2_6BD_Rx_Timer(IN := NOT(OrionBMS2_6BD_Rx.q_NewData), PT := T#3S);
IF (OrionBMS2_6B0_Rx_Timer.Q = TRUE AND OrionBMS2_6B1_Rx_Timer.Q = TRUE AND OrionBMS2_6B2_Rx_Timer.Q = TRUE AND
	OrionBMS2_6B3_Rx_Timer.Q = TRUE AND OrionBMS2_6B4_Rx_Timer.Q = TRUE AND OrionBMS2_6B5_Rx_Timer.Q = TRUE AND
	OrionBMS2_6B6_Rx_Timer.Q = TRUE AND OrionBMS2_6B7_Rx_Timer.Q = TRUE AND OrionBMS2_6B8_Rx_Timer.Q = TRUE AND
	OrionBMS2_6B9_Rx_Timer.Q = TRUE AND OrionBMS2_6BA_Rx_Timer.Q = TRUE AND OrionBMS2_6BB_Rx_Timer.Q = TRUE AND
	OrionBMS2_6BC_Rx_Timer.Q = TRUE AND OrionBMS2_6BD_Rx_Timer.Q = TRUE											) THEN

	gq_OrionBMS2_CommsLoss	:=	TRUE;
ELSE
	gq_OrionBMS2_CommsLoss	:=	FALSE;
END_IF


OrionBMS2_RxConversion();

END_PROGRAM

// Application/UserCode/BMS/OrionBMS/OrionBMS2_RxConversion_1
PROGRAM OrionBMS2_RxConversion_1
VAR
	(**********************************************************)
	(*Rx Conversion*)
	gr_OrionBMS2_PackVoltage			:	REAL;
	gr_OrionBMS2_PackCurrent			:	REAL;
	gr_OrionBMS2_PackSOC				:	REAL;
	gr_OrionBMS2_Max_Charging_Voltage	:	REAL;
	gq_BMS2_BalActive			:BOOL;
	gq_BMS2_Flag_1				:BOOL;
	gq_BMS2_Flag_2				:BOOL;
	gq_BMS2_Flag_3				:BOOL;
	gq_BMS2_Flag_4				:BOOL;
	gq_BMS2_Flag_5				:BOOL;
	gq_BMS2_Flag_6				:BOOL;
	gq_BMS2_Flag_7				:BOOL;
	Safety_OK   : BOOL;
END_VAR
VAR CONSTANT
	SYSTEMRX_CF	:	REAL	:=	0.1;
	CURRENT_CF	:	REAL	:=	0.1;
END_VAR

(*Convert input variables into real units by applying conversion factors and offsets*)

gr_OrionBMS2_PackVoltage			:=	UINT_TO_REAL(gu16_OrionBMS2_PackVoltage) * SYSTEMRX_CF;
gr_OrionBMS2_PackCurrent			:=	INT_TO_REAL(gs16_OrionBMS2_PackCurrent) * CURRENT_CF;
gr_OrionBMS2_PackSOC				:=	REAL_TO_USINT(gu8_OrionBMS2_RAW_SOC / 2);
gr_OrionBMS2_Max_Charging_Voltage	:= gu8_OrionBMS2_PopulatedCells *3.65;
	
OrionBMS2_DTCFlag1_0A07_DischargeLimitEnforcementFault		:=	gu16_OrionBMS2_DTC_Flags1.0;
OrionBMS2_DTCFlag1_0A08_ChargerSafetyRelayFault 			:=	gu16_OrionBMS2_DTC_Flags1.1;
OrionBMS2_DTCFlag1_0A09_InternalHardwareFault				:=	gu16_OrionBMS2_DTC_Flags1.2;
OrionBMS2_DTCFlag1_0A0A_InternalHeatskinkThermistorFault 	:=	gu16_OrionBMS2_DTC_Flags1.3;
OrionBMS2_DTCFlag1_0A0B_InternalSoftwareFault				:=	gu16_OrionBMS2_DTC_Flags1.4;
OrionBMS2_DTCFlag1_0A0C_HighestCellVoltageTooHighFault 	:=	gu16_OrionBMS2_DTC_Flags1.5;
OrionBMS2_DTCFlag1_0A0E_LowestCellVoltageTooLowFault 		:=	gu16_OrionBMS2_DTC_Flags1.6;
OrionBMS2_DTCFlag1_0A10_PackTooHotFault 					:=	gu16_OrionBMS2_DTC_Flags1.7;
OrionBMS2_DTCFlags_Reserved_Bit8 							:=	gu16_OrionBMS2_DTC_Flags1.8;
OrionBMS2_DTCFlags_Reserved_Bit9 							:=	gu16_OrionBMS2_DTC_Flags1.9;
OrionBMS2_DTCFlags_Reserved_Bit10 							:=	gu16_OrionBMS2_DTC_Flags1.10;
OrionBMS2_DTCFlags_Reserved_Bit11 							:=	gu16_OrionBMS2_DTC_Flags1.11;
OrionBMS2_DTCFlags_Reserved_Bit12 							:=	gu16_OrionBMS2_DTC_Flags1.12;
OrionBMS2_DTCFlags_Reserved_Bit13 							:=	gu16_OrionBMS2_DTC_Flags1.13;
OrionBMS2_DTCFlags_Reserved_Bit14 							:=	gu16_OrionBMS2_DTC_Flags1.14;
OrionBMS2_DTCFlags_Reserved_Bit15							:=	gu16_OrionBMS2_DTC_Flags1.15;

OrionBMS2_DTCFlags2_0A1F_InternalCommunicationFault			:=	gu16_OrionBMS2_DTC_Flags2.8;
OrionBMS2_DTCFlags2_0A12_CellBalancingStruckOffFault		:=	gu16_OrionBMS2_DTC_Flags2.9;
OrionBMS2_DTCFlags2_0A80_WeakCellFault						:=	gu16_OrionBMS2_DTC_Flags2.10;
OrionBMS2_DTCFlags2_0AFA_LowCellVoltageFault				:=	gu16_OrionBMS2_DTC_Flags2.11;
OrionBMS2_DTCFlags2_0A04_OpenWiringFault					:=	gu16_OrionBMS2_DTC_Flags2.12;
OrionBMS2_DTCFlags2_0AC0_CurrentSensorFault					:=	gu16_OrionBMS2_DTC_Flags2.13;
OrionBMS2_DTCFlags2_0A0D_HighestCellVoltageOver5vFault		:=	gu16_OrionBMS2_DTC_Flags2.14;
OrionBMS2_DTCFlags2_0A0F_CellASICFault						:=	gu16_OrionBMS2_DTC_Flags2.15;
OrionBMS2_DTCFlags2_0A02_WeakPackFault						:=	gu16_OrionBMS2_DTC_Flags2.0;
OrionBMS2_DTCFlags2_0A81_FanMonitorFault					:=	gu16_OrionBMS2_DTC_Flags2.1;
OrionBMS2_DTCFlags2_0A9C_ThermistorFault					:=	gu16_OrionBMS2_DTC_Flags2.2;
OrionBMS2_DTCFlags2_0100_ExternalCommunicationFault			:=	gu16_OrionBMS2_DTC_Flags2.3;
OrionBMS2_DTCFlags2_0560_RedundantPowerSupplyFault			:=	gu16_OrionBMS2_DTC_Flags2.4;
OrionBMS2_DTCFlags2_0AA6_HighVoltageIsolatonFault			:=	gu16_OrionBMS2_DTC_Flags2.5;
OrionBMS2_DTCFlags2_0A05_InputPowerSupplyFault				:=	gu16_OrionBMS2_DTC_Flags2.6;
OrionBMS2_DTCFlags2_0A06_ChargeLimitEnforcementFault		:=	gu16_OrionBMS2_DTC_Flags2.7;	
	
gq_BMS2_BalActive			:=	gu8_OrionBMS2_Custom_Flag_1.0;
gq_BMS2_Flag_1				:=	gu8_OrionBMS2_Custom_Flag_1.1;
gq_BMS2_Flag_2				:=	gu8_OrionBMS2_Custom_Flag_1.2;
gq_BMS2_Flag_3				:=	gu8_OrionBMS2_Custom_Flag_1.3;
gq_BMS2_Flag_4				:=	gu8_OrionBMS2_Custom_Flag_1.4;
gq_BMS2_Flag_5				:=	gu8_OrionBMS2_Custom_Flag_1.5;
gq_BMS2_Flag_6				:=	gu8_OrionBMS2_Custom_Flag_1.6;
Safety_OK    				:=	gu8_OrionBMS2_Custom_Flag_1.7;

END_PROGRAM

// Application/UserCode/BMS/OrionBMS/OrionBMS_Tx_1
PROGRAM OrionBMS_Tx_1
VAR
	ht_OrionBMS1_State_Tx	:	EPEC_CANVXD.Msg;
	ht_OrionBMS2_State_Tx	:	EPEC_CANVXD.Msg;
	hton_MessageSend_Timer	:	TON;
END_VAR

(*Transmit control of both BMS*)

(*Setup output message structure with ID, Data and Length*)
ht_OrionBMS1_State_Tx.ID	:=	16#023;
ht_OrionBMS1_State_Tx.Data[0]	:=	gu8_BMS1_MPO_1_State;
ht_OrionBMS1_State_Tx.Data[1]	:=	gu8_BMS1_MPO_2_State;
ht_OrionBMS1_State_Tx.Data[2]	:=	gu8_BMS1_MPO_3_State;
ht_OrionBMS1_State_Tx.Data[3]	:=	gu8_BMS1_MPO_4_State;
ht_OrionBMS1_State_Tx.Data[4]	:=	gu8_BMS1_MPE_State;
ht_OrionBMS1_State_Tx.Data[5]	:=	0;
ht_OrionBMS1_State_Tx.Data[6]	:=	0;
ht_OrionBMS1_State_Tx.Data[7]	:=	0;
ht_OrionBMS1_State_Tx.Len	:=	8;

(*Setup output message structure with ID, Data and Length*)
ht_OrionBMS2_State_Tx.ID	:=	16#023;
ht_OrionBMS2_State_Tx.Data[0]	:=	gu8_BMS2_MPO_1_State;
ht_OrionBMS2_State_Tx.Data[1]	:=	gu8_BMS2_MPO_2_State;
ht_OrionBMS2_State_Tx.Data[2]	:=	gu8_BMS2_MPO_3_State;
ht_OrionBMS2_State_Tx.Data[3]	:=	gu8_BMS2_MPO_4_State;
ht_OrionBMS2_State_Tx.Data[4]	:=	gu8_BMS2_MPE_State;
ht_OrionBMS2_State_Tx.Data[5]	:=	0;
ht_OrionBMS2_State_Tx.Data[6]	:=	0;
ht_OrionBMS2_State_Tx.Data[7]	:=	0;
ht_OrionBMS2_State_Tx.Len	:=	8;

(*Same message needed for both BMS so structure for BMS1 saved across into BMS2   NOW SEPERATE!!*)
(*ht_OrionBMS2_State_Tx	:=	ht_OrionBMS1_State_Tx;*)

(*Message broadcast timer and actual structure send on CANbus*)
hton_MessageSend_Timer(IN := NOT(hton_MessageSend_Timer.Q), PT := T#100MS);
IF (hton_MessageSend_Timer.Q = TRUE) THEN
	G_CAN2_Channel.SendMessage(i_pMSG:=ADR(ht_OrionBMS1_State_Tx));
	G_CAN3_Channel.SendMessage(i_pMSG:=ADR(ht_OrionBMS2_State_Tx));
END_IF

END_PROGRAM

// Application/UserCode/Brusa/Brusa1_Comms/Brusa1_Rx_1
PROGRAM Brusa1_Rx_1
VAR
	ActAC_Rx			:	Receive_CAN2_STD;
	ActErr_Rx			:	Receive_CAN2_STD;
	ActInt_Rx			:	Receive_CAN2_STD;
	ActLim_Rx			:	Receive_CAN2_STD;
	ActPlug_Rx			:	Receive_CAN2_STD;
	
	ActAC_Rx_Timer		:	TON;
	ActErr_Rx_Timer		:	TON;
	ActInt_Rx_Timer		:	TON;
	ActLim_Rx_Timer		:	TON;
	ActPlug_Rx_Timer	:	TON;
	
	StatusPP_Rx			:	USINT; 
	StatusPP_Prev		:	USINT;
	
	ACVoltL1Act_Rx		:	USINT;
	ACVoltL2Act_Rx		:	USINT;
	ACVoltL3Act_Rx		:	USINT;
	ACFreqAct			:	USINT;
	SACPhaseRot			:	BOOL;
	ACCurrL1Act_Rx		:	USINT;
	ACCurrL2Act_Rx		:	USINT;
	ACCurrL3Act_Rx		:	USINT;
	ACPowTotAct_Rx		:	USINT;
	
	(*Act Err*)
	E_WrongHW			: BOOL;
	E_WrongFPGA			: BOOL;
	E_EPGAInit			: BOOL;
	E_NVSRam			: BOOL;
	E_Flash				: BOOL;
	E_OSTrap			: BOOL;
	E_HVIsoPos			: BOOL;
	E_HVIsoNeg			: BOOL;
	E_Internal			: BOOL;
	E_TempInt			: BOOL;
	E_DCHVVoltRed		: BOOL;
	E_IntSupply			: BOOL;
	E_CANMsgLost		: BOOL;
	E_CANValue			: BOOL;
	E_ACInterruption	: BOOL;
	E_DCHVVoltRange		: BOOL;
	E_TempCon			: BOOL;
	E_ConLocked			: BOOL;
	E_Interlock			: BOOL;
	E_Crash				: BOOL;
	E_PRELOAD			: BOOL;
	E_BURST				: BOOL;
	E_TPON				: BOOL;
	E_UZK				: BOOL;
	E_LatchFPGA			: BOOL;
	E_OverTemp			: BOOL;
	(*Warnings*)
	W_Watchdog			: BOOL;
	W_PowRed			: BOOL;
	W_TempInt			: BOOL;
	W_CANTimeout		: BOOL;
	W_CANOff			: BOOL;
	W_CANRx				: BOOL;
	W_CANTx				: BOOL;
	W_ConLocked			: BOOL;
	W_FPGA				: BOOL;
	W_ACVoltage			: BOOL;
	W_ACFrequency		: BOOL;
	W_PRELOAD			: BOOL;
	
	(*Act Int*)
	ACWhAct				:	UINT;
	DCHVWhAct			:	UINT;
	MaxTempAct_Rx		:	USINT;
	TempCon_Rx			:	USINT;
	DCHVAhAct_Rx		:	UINT;
	(*Act Lim*)
	StateCrtlPilot		:	USINT;
	DCHVVoltAct_Rx		:	UINT;
	StateAct			:	USINT; //0:Sleep 1:Wakeup 2:Standby 3:Ready2Charge 4:Charge 5:Shutdown
	S_DCHVCurrLim		:	BOOL;
	S_DCHVVoltLim		:	BOOL;
	DCHVCurrAct_Rx		:	UINT;
	S_ProximityLim		:	BOOL;
	S_CtrlPilotLim		:	BOOL;
	S_ConTempLim		:	BOOL;
	S_IntTempLim		:	BOOL;
	S_ACCurrLim			:	BOOL;
	ACCurrMaxAct_Rx		:	UINT;
	ACCurrHWAvl_Rx		:	USINT;
	S_ProximityDet		:	BOOL;
	S_CtrlPilotDet		:	BOOL;
	S_ConLocked			:	BOOL;
	S_ACDet				:	BOOL;
	S_HWWakeup			:	BOOL;
	S_HWEnablErre		:	BOOL;
	S_Err				:	BOOL;
	S_Warn				:	BOOL;
	(*Act Plug*)
	StatusCP			:	USINT;
	S_CPX1				:	BOOL;
	S_CPSCC				:	BOOL;
	ACCurrMaxCP_Rx		:	UINT;
	StatusPP			:	USINT; //0:PROXD_DETECTED 1:PROXD_CIRCUIT_RANGE 2:PROXD_CIRCUIT_LOW 3:PROXD_CIRCUIT_HIGH 4:PROXD_CIRCUIT_ERRATIC 5:PROXD_NOT_CONNECTED 7:SNA
	ACCurrMaxPP			:	USINT; //0:0 A 1:13 A 2:20 A 3:32 A 4:63 A 7:SNA
	s_ACVoltDerate		:	BOOL;
	S_ACDerating		:	BOOL;
	ACPhaseUsd			:	USINT;
	ACPhaseDet			:	USINT;  ///kak Why not used?????????
	CoolingRequest		:	USINT;
	TempCoolPlate_Rx	:	USINT; //Actual temperatur cool plate 255:SNA
	CommsLoss			:	BOOL;
	C_EnPhaseShift		:	BOOL;
END_VAR


ActAC_Rx(u32_COBID	:=	16#729,
				q_NewData => ,
				au8_Data => ,
				u8_Length => 			);
				
ActErr_Rx(u32_COBID	:=	16#799,
				q_NewData => ,
				au8_Data => ,
				u8_Length => 			);
				
ActInt_Rx(u32_COBID	:=	16#709,
				q_NewData => ,
				au8_Data => ,
				u8_Length => 			);
				
ActLim_Rx(u32_COBID	:=	16#728,
				q_NewData => ,
				au8_Data => ,
				u8_Length => 			);
				
ActPlug_Rx(u32_COBID	:=	16#739,
				q_NewData => ,
				au8_Data => ,
				u8_Length => 			);

(*Act AC*)
ACVoltL1Act_Rx		:=	ActAC_Rx.au8_Data[0];
ACVoltL2Act_Rx		:=	ActAC_Rx.au8_Data[1];
ACVoltL3Act_Rx		:=	ActAC_Rx.au8_Data[2];
ACFreqAct			:=	(ActAC_Rx.au8_Data[3] AND 2#01111111); (*Mask*)
SACPhaseRot			:=	ActAC_Rx.au8_Data[3].7;
ACCurrL1Act_Rx		:=	ActAC_Rx.au8_Data[4];
ACCurrL2Act_Rx		:=	ActAC_Rx.au8_Data[5];
ACCurrL3Act_Rx		:=	ActAC_Rx.au8_Data[6];
ACPowTotAct_Rx		:=	ActAC_Rx.au8_Data[7];;

(*Act Err*)
E_WrongHW			:=	ActErr_Rx.au8_Data[0].0;
E_WrongFPGA			:=	ActErr_Rx.au8_Data[0].1;
E_EPGAInit			:=	ActErr_Rx.au8_Data[0].2;
E_NVSRam			:=	ActErr_Rx.au8_Data[0].5;
E_Flash				:=	ActErr_Rx.au8_Data[0].6;
E_OSTrap			:=	ActErr_Rx.au8_Data[0].7;
E_HVIsoPos			:=	ActErr_Rx.au8_Data[1].1;
E_HVIsoNeg			:=	ActErr_Rx.au8_Data[1].2;
E_Internal			:=	ActErr_Rx.au8_Data[1].4;
E_TempInt			:=	ActErr_Rx.au8_Data[1].5;
E_DCHVVoltRed		:=	ActErr_Rx.au8_Data[1].6;
E_IntSupply			:=	ActErr_Rx.au8_Data[1].7;
E_CANMsgLost		:=	ActErr_Rx.au8_Data[2].0;
E_CANValue			:=	ActErr_Rx.au8_Data[2].1;
E_ACInterruption	:=	ActErr_Rx.au8_Data[2].2;
E_DCHVVoltRange		:=	ActErr_Rx.au8_Data[2].3;
E_TempCon			:=	ActErr_Rx.au8_Data[2].4;
E_ConLocked			:=	ActErr_Rx.au8_Data[2].5;
E_Interlock			:=	ActErr_Rx.au8_Data[2].6;
E_Crash				:=	ActErr_Rx.au8_Data[2].7;
E_PRELOAD			:=	ActErr_Rx.au8_Data[3].1;
E_BURST				:=	ActErr_Rx.au8_Data[3].2;
E_TPON				:=	ActErr_Rx.au8_Data[3].3;
E_UZK				:=	ActErr_Rx.au8_Data[3].4;
E_LatchFPGA			:=	ActErr_Rx.au8_Data[3].5;
E_OverTemp			:=	ActErr_Rx.au8_Data[3].7;
W_Watchdog			:=	ActErr_Rx.au8_Data[4].7;
W_PowRed			:=	ActErr_Rx.au8_Data[5].0;
W_TempInt			:=	ActErr_Rx.au8_Data[5].1;
W_CANTimeout		:=	ActErr_Rx.au8_Data[6].0;
W_CANOff			:=	ActErr_Rx.au8_Data[6].1;
W_CANRx				:=	ActErr_Rx.au8_Data[6].2;
W_CANTx				:=	ActErr_Rx.au8_Data[6].3;
W_ConLocked			:=	ActErr_Rx.au8_Data[6].7;
W_FPGA				:=	ActErr_Rx.au8_Data[7].0;
W_ACVoltage			:=	ActErr_Rx.au8_Data[7].1;
W_ACFrequency		:=	ActErr_Rx.au8_Data[7].2;
W_PRELOAD			:=	ActErr_Rx.au8_Data[7].3;


(*Act Int*)
ACWhAct			:=	SHL(USINT_TO_UINT(ActInt_Rx.au8_Data[0]), 8) +
								USINT_TO_UINT(ActInt_Rx.au8_Data[1]);
DCHVWhAct			:=	SHL(USINT_TO_UINT(ActInt_Rx.au8_Data[2]), 8) +
								USINT_TO_UINT(ActInt_Rx.au8_Data[3]);
MaxTempAct_Rx		:=	ActInt_Rx.au8_Data[4];
TempCon_Rx			:=	ActInt_Rx.au8_Data[5];
DCHVAhAct_Rx		:=	SHL(USINT_TO_UINT(ActInt_Rx.au8_Data[6]), 8) +
								USINT_TO_UINT(ActInt_Rx.au8_Data[7]);
(*Act Lim*)
StateCrtlPilot		:=	SHR((ActLim_Rx.au8_Data[0] AND 2#11100000), 5);
DCHVVoltAct_Rx	:=	SHL(USINT_TO_UINT(ActLim_Rx.au8_Data[0] AND 2#00011111), 8) +
								USINT_TO_UINT(ActLim_Rx.au8_Data[1]);
StateAct			:=	SHR((ActLim_Rx.au8_Data[2] AND 2#11100000), 5);
S_DCHVCurrLim		:=	ActLim_Rx.au8_Data[2].4;
S_DCHVVoltLim		:=	ActLim_Rx.au8_Data[2].3;
DCHVCurrAct_Rx	:=	SHL(USINT_TO_UINT(ActLim_Rx.au8_Data[2] AND 2#00000111), 8) +
								USINT_TO_UINT(ActLim_Rx.au8_Data[3]);
S_ProximityLim		:=	ActLim_Rx.au8_Data[4].7;
S_CtrlPilotLim		:=	ActLim_Rx.au8_Data[4].6;
S_ConTempLim		:=	ActLim_Rx.au8_Data[4].5;
S_IntTempLim		:=	ActLim_Rx.au8_Data[4].4;
S_ACCurrLim			:=	ActLim_Rx.au8_Data[4].3;
ACCurrMaxAct_Rx	:=	SHL(USINT_TO_UINT(ActLim_Rx.au8_Data[4] AND 2#00000111), 8) +
								USINT_TO_UINT(ActLim_Rx.au8_Data[5]);
ACCurrHWAvl_Rx		:=	ActLim_Rx.au8_Data[6];
S_ProximityDet		:=	ActLim_Rx.au8_Data[7].7;
S_CtrlPilotDet		:=	ActLim_Rx.au8_Data[7].6;
S_ConLocked			:=	ActLim_Rx.au8_Data[7].5;
S_ACDet				:=	ActLim_Rx.au8_Data[7].4;
S_HWWakeup			:=	ActLim_Rx.au8_Data[7].3;
S_HWEnablErre		:=	ActLim_Rx.au8_Data[7].2;
S_Err				:=	ActLim_Rx.au8_Data[7].1;
S_Warn				:=	ActLim_Rx.au8_Data[7].0;
(*Act Plug*)
StatusCP			:=	ActPlug_Rx.au8_Data[0] AND 2#11100000;
S_CPX1				:=	ActPlug_Rx.au8_Data[0].4;
S_CPSCC				:=	ActPlug_Rx.au8_Data[0].3;
ACCurrMaxCP_Rx	:=	SHL(USINT_TO_UINT(ActPlug_Rx.au8_Data[0] AND 2#00000011), 8) +
								USINT_TO_UINT(ActPlug_Rx.au8_Data[1]);
StatusPP_Rx			:=	SHR((ActPlug_Rx.au8_Data[2] AND 2#01110000), 4);
ACCurrMaxPP		:=	ActPlug_Rx.au8_Data[2] AND 2#00001111;
s_ACVoltDerate		:=	ActPlug_Rx.au8_Data[4].7;
S_ACDerating		:=	ActPlug_Rx.au8_Data[4].6;
ACPhaseUsd			:=	SHR((ActPlug_Rx.au8_Data[4] AND 2#00111000), 3);
ACPhaseDet			:=	ActPlug_Rx.au8_Data[4] AND 2#00000111;
CoolingRequest		:=	ActPlug_Rx.au8_Data[5] AND 2#01111111;
TempCoolPlate_Rx	:=	ActPlug_Rx.au8_Data[6];


IF NOT(Brusa1_Tx.hton_NoPP_StopTx_Timer.Q) THEN
	ActAC_Rx_Timer(IN := NOT(ActAC_Rx.q_NewData), PT := T#5S);
	ActErr_Rx_Timer(IN := NOT(ActErr_Rx.q_NewData), PT := T#5S);
	ActInt_Rx_Timer(IN := NOT(ActInt_Rx.q_NewData), PT := T#5S);
	ActLim_Rx_Timer(IN := NOT(ActLim_Rx.q_NewData), PT := T#5S);
	ActPlug_Rx_Timer(IN := NOT(ActPlug_Rx.q_NewData), PT := T#5S);
	
	IF (ActAC_Rx_Timer.Q AND ActErr_Rx_Timer.Q AND ActInt_Rx_Timer.Q AND
		ActLim_Rx_Timer.Q AND ActPlug_Rx_Timer.Q) THEN
		CommsLoss	:=	TRUE;
	ELSE
		CommsLoss	:=	FALSE;
	END_IF
END_IF

(*Only update Status PP if both this value and the previous value are the same*)
IF (StatusPP_Rx = StatusPP_Prev) THEN
	StatusPP	:=	StatusPP_Rx;
END_IF
StatusPP_Prev	:=	StatusPP_Rx;

Brusa1_RxConversion();

END_PROGRAM

// Application/UserCode/Brusa/Brusa1_Comms/Brusa1_RxConversion_1
PROGRAM Brusa1_RxConversion_1
VAR
	ACVoltL1Act		:	UINT;
	ACVoltL2Act		:	UINT;
	ACVoltL3Act		:	UINT;
	ACCurrL1Act		:	SINT;
	ACCurrL2Act		:	SINT;
	ACCurrL3Act		:	SINT;
	ACPowTotAct		:	UINT;
	MaxTempAct		:	INT;
	TempCon			:	INT;
	DCHVAhAct		:	REAL;
	DCHVVoltAct		:	REAL;
	DCHVCurrAct		:	REAL;
	ACCurrMaxAct	:	REAL;
	ACCurrHWAvl		:	REAL;
	ACCurrMaxCP		:	REAL;
	TempCoolPlate	:	INT;	
END_VAR

ACVoltL1Act	:=	USINT_TO_UINT(Brusa1_Rx.ACVoltL1Act_Rx) * 2;
ACVoltL2Act	:=	USINT_TO_UINT(Brusa1_Rx.ACVoltL2Act_Rx) * 2;
ACVoltL3Act	:=	USINT_TO_UINT(Brusa1_Rx.ACVoltL3Act_Rx) * 2;
ACCurrL1Act	:=	USINT_TO_SINT(Brusa1_Rx.ACCurrL1Act_Rx) - 127;
ACCurrL2Act	:=	USINT_TO_SINT(Brusa1_Rx.ACCurrL2Act_Rx) - 127;
ACCurrL3Act	:=	USINT_TO_SINT(Brusa1_Rx.ACCurrL3Act_Rx) - 127;
ACPowTotAct	:=	USINT_TO_UINT(Brusa1_Rx.ACPowTotAct_Rx) * 100;
MaxTempAct	:=	USINT_TO_INT(Brusa1_Rx.MaxTempAct_Rx) - 50;
TempCon		:=	USINT_TO_INT(Brusa1_Rx.TempCon_Rx) - 50;
DCHVAhAct		:=	UINT_TO_REAL(Brusa1_Rx.DCHVAhAct_Rx) * 0.01;
DCHVVoltAct		:=	UINT_TO_REAL(Brusa1_Rx.DCHVVoltAct_Rx) * 0.1;
DCHVCurrAct		:=	UINT_TO_REAL(Brusa1_Rx.DCHVCurrAct_Rx) * 0.1 - 100;
ACCurrMaxAct	:=	UINT_TO_REAL(Brusa1_Rx.ACCurrMaxAct_Rx) * 0.1 -100;
ACCurrHWAvl		:=	USINT_TO_REAL(Brusa1_Rx.ACCurrHWAvl_Rx) * 0.5;
ACCurrMaxCP		:=	UINT_TO_REAL(Brusa1_Rx.ACCurrMaxCP_Rx) * 0.1;
TempCoolPlate	:=	USINT_TO_INT(Brusa1_Rx.TempCoolPlate_Rx) - 50;

END_PROGRAM

// Application/UserCode/Brusa/Brusa1_Comms/Brusa1_Tx_1
PROGRAM Brusa1_Tx_1
VAR
	DenLim_Tx				:	EPEC_CANVXD.Msg;
	hu8_DenLim_Tx0			:	BYTE;
	hu8_DenLim_Tx2			:	BYTE;
	hu8_DenLim_Tx4			:	BYTE;
	hu8_DenLim_Tx6			:	BYTE;
	hton_Transmit_Timer		:	TON;
	hton_NoPP_StopTx_Timer	:	TON;
	StopBroadcast			:	BOOL;
	C_VentilRq				: 	BOOL;
END_VAR

//r2

Brusa1_TxConversion();

StopBroadcast	:=	(NOT(Brusa1_Rx.S_ProximityDet)(* AND DI_q_VehicleKL15_DI = FALSE*));
hton_NoPP_StopTx_Timer(IN := StopBroadcast, PT := T#1S);

// Brusa1_Control.C_Clr_Err	:= FALSE; 

hu8_DenLim_Tx0	        :=	UINT_TO_USINT(SHR(Brusa1_TxConversion.DCHVVoltLimMax_Tx, 8)) + SHL(BOOL_TO_USINT(C_VentilRq), 5) +
					        SHL(BOOL_TO_USINT(Brusa.M_Unlock), 6) + SHL(BOOL_TO_USINT((*Brusa.M_ErrCLr*) FALSE), 7);
hu8_DenLim_Tx2	        :=	(UINT_TO_USINT(SHR(Brusa1_TxConversion.DCHVCurrLimMax_Tx, 8)) AND 2#00000111) + SHL(Brusa.M_StateDem, 5);
hu8_DenLim_Tx4	        :=	(UINT_TO_USINT(SHR(Brusa1_TxConversion.ACCurrLimMax_Tx, 8)) AND 2#00000111) + SHL(Brusa.LEDDem, 4);
//hu8_DenLim_Tx6	        :=	(UINT_TO_USINT(SHR(Brusa1_TxConversion.ACPhaseShift_Tx, 8)) AND 2#00001111) + SHL(BOOL_TO_USINT(Brusa1_Rx.C_EnPhaseShift), 4); //kak ac or en??????????????????????????

DenLim_Tx.ID		:=	16#711;
DenLim_Tx.Data[0]	:=	hu8_DenLim_Tx0;
DenLim_Tx.Data[1]	:=	UINT_TO_USINT(Brusa1_TxConversion.DCHVVoltLimMax_Tx);
DenLim_Tx.Data[2]	:=	hu8_DenLim_Tx2;
DenLim_Tx.Data[3]	:=	UINT_TO_USINT(Brusa1_TxConversion.DCHVCurrLimMax_Tx);
DenLim_Tx.Data[4]	:=	hu8_DenLim_Tx4;
DenLim_Tx.Data[5]	:=	UINT_TO_USINT(Brusa1_TxConversion.ACCurrLimMax_Tx);
DenLim_Tx.Data[6]	:=	hu8_DenLim_Tx6;
DenLim_Tx.Data[7]	:=	UINT_TO_USINT(Brusa1_TxConversion.ACPhaseShift_Tx);
DenLim_Tx.Len		:=	8;


hton_Transmit_Timer(IN := NOT(hton_Transmit_Timer.Q), PT := T#90MS);
IF (hton_Transmit_Timer.Q = TRUE AND NOT(hton_NoPP_StopTx_Timer.Q) = TRUE) THEN
	G_CAN2_Channel.SendMessage(i_pMSG:=ADR(DenLim_Tx));
END_IF

END_PROGRAM

// Application/UserCode/Brusa/Brusa1_Comms/Brusa1_TxConversion_1
PROGRAM Brusa1_TxConversion_1
VAR
		DCHVVoltLimMax_Tx	:	UINT;
		DCHVCurrLimMax_Tx	:	UINT;
		ACCurrLimMax_Tx		:	UINT;
		ACPhaseShift_Tx		:	UINT;
END_VAR


DCHVVoltLimMax_Tx	:=	REAL_TO_UINT(Brusa.M_DCHVVoltLimMax / 0.1);
DCHVCurrLimMax_Tx	:=	REAL_TO_UINT((Brusa.M_DCHVCurrLimMax - 102.4) / 0.1);
ACCurrLimMax_Tx		:=	REAL_TO_UINT((Brusa.M_ACCurrLimMax - 102.4) / 0.1);
//ACPhaseShift_Tx		:=	REAL_TO_UINT(Brusa1_Control.ACPhaseShift / 0.1);

END_PROGRAM

// Application/UserCode/Brusa/Brusa2_Comms/Brusa2_Rx_1
PROGRAM Brusa2_Rx_1
VAR
	ActAC_Rx	:	Receive_CAN3_STD;
	NLG2_ActErr_Rx	:	Receive_CAN3_STD;
	NLG2_ActInt_Rx	:	Receive_CAN3_STD;
	NLG2_ActLim_Rx	:	Receive_CAN3_STD;
	NLG2_ActPlug_Rx	:	Receive_CAN3_STD;
	
	ActAC_Rx_Timer		:	TON;
	ActErr_Rx_Timer		:	TON;
	ActInt_Rx_Timer		:	TON;
	ActLim_Rx_Timer		:	TON;
	ActPlug_Rx_Timer	:	TON;
	
	StatusPP_Rx			:	USINT; 
	StatusPP_Prev		:	USINT;
	
	ACVoltL1Act_Rx		:	USINT;
	ACVoltL2Act_Rx		:	USINT;
	ACVoltL3Act_Rx		:	USINT;
	ACFreqAct			:	USINT;
	SACPhaseRot			:	BOOL;
	ACCurrL1Act_Rx		:	USINT;
	ACCurrL2Act_Rx		:	USINT;
	ACCurrL3Act_Rx		:	USINT;
	ACPowTotAct_Rx		:	USINT;
	
	(*Act Err*)
	E_WrongHW					: BOOL;
	E_WrongFPGA					: BOOL;
	E_EPGAInit					: BOOL;
	E_NVSRam					: BOOL;
	E_Flash						: BOOL;
	E_OSTrap					: BOOL;
	E_HVIsoPos			: BOOL;
	E_HVIsoNeg			: BOOL;
	E_Internal			: BOOL;
	E_TempInt			: BOOL;
	E_DCHVVoltRed		: BOOL;
	E_IntSupply			: BOOL;
	E_CANMsgLost		: BOOL;
	E_CANValue			: BOOL;
	E_ACInterruption	: BOOL;
	E_DCHVVoltRange		: BOOL;
	E_TempCon			: BOOL;
	E_ConLocked			: BOOL;
	E_Interlock			: BOOL;
	E_Crash				: BOOL;
	E_PRELOAD			: BOOL;
	E_BURST				: BOOL;
	E_TPON				: BOOL;
	E_UZK				: BOOL;
	E_LatchFPGA					: BOOL;
	E_OverTemp					: BOOL;
	(*Warnings*)
	W_Watchdog					: BOOL;
	W_PowRed			: BOOL;
	W_TempInt			: BOOL;
	W_CANTimeout		: BOOL;
	W_CANOff			: BOOL;
	W_CANRx				: BOOL;
	W_CANTx				: BOOL;
	W_ConLocked			: BOOL;
	W_FPGA				: BOOL;
	W_ACVoltage			: BOOL;
	W_ACFrequency		: BOOL;
	W_PRELOAD			: BOOL;
	
	(*Act Int*)
	ACWhAct			:	UINT;
	DCHVWhAct			:	UINT;
	MaxTempAct_Rx		:	USINT;
	TempCon_Rx					:	USINT;
	DCHVAhAct_Rx				:	UINT;
	(*Act Lim*)
	StateCrtlPilot				:	USINT;
	DCHVVoltAct_Rx				:	UINT;
	StateAct					:	USINT; //0:Sleep 1:Wakeup 2:Standby 3:Ready2Charge 4:Charge 5:Shutdown
	S_DCHVCurrLim				:	BOOL;
	S_DCHVVoltLim				:	BOOL;
	DCHVCurrAct_Rx	:	UINT;
	S_ProximityLim		:	BOOL;
	S_CtrlPilotLim		:	BOOL;
	S_ConTempLim		:	BOOL;
	S_IntTempLim		:	BOOL;
	S_ACCurrLim			:	BOOL;
	ACCurrMaxAct_Rx		:	UINT;
	ACCurrHWAvl_Rx		:	USINT;
	S_ProximityDet		:	BOOL;
	S_CtrlPilotDet		:	BOOL;
	S_ConLocked			:	BOOL;
	S_ACDet				:	BOOL;
	S_HWWakeup			:	BOOL;
	S_HWEnablErre		:	BOOL;
	S_Err				:	BOOL;
	S_Warn				:	BOOL;
	(*Act Plug*)
	StatusCP			:	USINT;
	S_CPX1					:	BOOL;
	S_CPSCC				:	BOOL;
	ACCurrMaxCP_Rx	:	UINT;
	StatusPP			:	USINT; //0:PROXD_DETECTED 1:PROXD_CIRCUIT_RANGE 2:PROXD_CIRCUIT_LOW 3:PROXD_CIRCUIT_HIGH 4:PROXD_CIRCUIT_ERRATIC 5:PROXD_NOT_CONNECTED 7:SNA
	ACCurrMaxPP			:	USINT; //0:0 A 1:13 A 2:20 A 3:32 A 4:63 A 7:SNA
	s_ACVoltDerate		:	BOOL;
	S_ACDerating		:	BOOL;
	ACPhaseUsd			:	USINT;
	ACPhaseDet			:	USINT;  ///kak Why not used?????????
	CoolingRequest		:	USINT;
	TempCoolPlate_Rx	:	USINT; //Actual temperatur cool plate 255:SNA
	CommsLoss					:	BOOL;
	C_EnPhaseShift				:	BOOL;
END_VAR



ActAC_Rx(u32_COBID	:=	16#729,
				q_NewData => ,
				au8_Data => ,
				u8_Length => 			);
				
NLG2_ActErr_Rx(u32_COBID	:=	16#799,
				q_NewData => ,
				au8_Data => ,
				u8_Length => 			);
				
NLG2_ActInt_Rx(u32_COBID	:=	16#709,
				q_NewData => ,
				au8_Data => ,
				u8_Length => 			);
				
NLG2_ActLim_Rx(u32_COBID	:=	16#728,
				q_NewData => ,
				au8_Data => ,
				u8_Length => 			);
				
NLG2_ActPlug_Rx(u32_COBID	:=	16#739,
				q_NewData => ,
				au8_Data => ,
				u8_Length => 			);

(*Act AC*)
ACVoltL1Act_Rx		:=	ActAC_Rx.au8_Data[0];
ACVoltL2Act_Rx		:=	ActAC_Rx.au8_Data[1];
ACVoltL3Act_Rx		:=	ActAC_Rx.au8_Data[2];
ACFreqAct			:=	(ActAC_Rx.au8_Data[3] AND 2#01111111); (*Mask*)
SACPhaseRot			:=	ActAC_Rx.au8_Data[3].7;
ACCurrL1Act_Rx		:=	ActAC_Rx.au8_Data[4];
ACCurrL2Act_Rx		:=	ActAC_Rx.au8_Data[5];
ACCurrL3Act_Rx		:=	ActAC_Rx.au8_Data[6];
ACPowTotAct_Rx		:=	ActAC_Rx.au8_Data[7];;

(*Act Err*)
E_WrongHW			:=	NLG2_ActErr_Rx.au8_Data[0].0;
E_WrongFPGA			:=	NLG2_ActErr_Rx.au8_Data[0].1;
E_EPGAInit			:=	NLG2_ActErr_Rx.au8_Data[0].2;
E_NVSRam			:=	NLG2_ActErr_Rx.au8_Data[0].5;
E_Flash				:=	NLG2_ActErr_Rx.au8_Data[0].6;
E_OSTrap			:=	NLG2_ActErr_Rx.au8_Data[0].7;
E_HVIsoPos			:=	NLG2_ActErr_Rx.au8_Data[1].1;
E_HVIsoNeg			:=	NLG2_ActErr_Rx.au8_Data[1].2;
E_Internal			:=	NLG2_ActErr_Rx.au8_Data[1].4;
E_TempInt			:=	NLG2_ActErr_Rx.au8_Data[1].5;
E_DCHVVoltRed		:=	NLG2_ActErr_Rx.au8_Data[1].6;
E_IntSupply			:=	NLG2_ActErr_Rx.au8_Data[1].7;
E_CANMsgLost		:=	NLG2_ActErr_Rx.au8_Data[2].0;
E_CANValue			:=	NLG2_ActErr_Rx.au8_Data[2].1;
E_ACInterruption	:=	NLG2_ActErr_Rx.au8_Data[2].2;
E_DCHVVoltRange		:=	NLG2_ActErr_Rx.au8_Data[2].3;
E_TempCon			:=	NLG2_ActErr_Rx.au8_Data[2].4;
E_ConLocked			:=	NLG2_ActErr_Rx.au8_Data[2].5;
E_Interlock			:=	NLG2_ActErr_Rx.au8_Data[2].6;
E_Crash				:=	NLG2_ActErr_Rx.au8_Data[2].7;
E_PRELOAD			:=	NLG2_ActErr_Rx.au8_Data[3].1;
E_BURST				:=	NLG2_ActErr_Rx.au8_Data[3].2;
E_TPON				:=	NLG2_ActErr_Rx.au8_Data[3].3;
E_UZK				:=	NLG2_ActErr_Rx.au8_Data[3].4;
E_LatchFPGA			:=	NLG2_ActErr_Rx.au8_Data[3].5;
E_OverTemp			:=	NLG2_ActErr_Rx.au8_Data[3].7;
W_Watchdog			:=	NLG2_ActErr_Rx.au8_Data[4].7;
W_PowRed			:=	NLG2_ActErr_Rx.au8_Data[5].0;
W_TempInt			:=	NLG2_ActErr_Rx.au8_Data[5].1;
W_CANTimeout		:=	NLG2_ActErr_Rx.au8_Data[6].0;
W_CANOff			:=	NLG2_ActErr_Rx.au8_Data[6].1;
W_CANRx				:=	NLG2_ActErr_Rx.au8_Data[6].2;
W_CANTx				:=	NLG2_ActErr_Rx.au8_Data[6].3;
W_ConLocked			:=	NLG2_ActErr_Rx.au8_Data[6].7;
W_FPGA				:=	NLG2_ActErr_Rx.au8_Data[7].0;
W_ACVoltage			:=	NLG2_ActErr_Rx.au8_Data[7].1;
W_ACFrequency		:=	NLG2_ActErr_Rx.au8_Data[7].2;
W_PRELOAD			:=	NLG2_ActErr_Rx.au8_Data[7].3;


(*Act Int*)
ACWhAct			:=	SHL(USINT_TO_UINT(NLG2_ActInt_Rx.au8_Data[0]), 8) +
								USINT_TO_UINT(NLG2_ActInt_Rx.au8_Data[1]);
DCHVWhAct			:=	SHL(USINT_TO_UINT(NLG2_ActInt_Rx.au8_Data[2]), 8) +
								USINT_TO_UINT(NLG2_ActInt_Rx.au8_Data[3]);
MaxTempAct_Rx		:=	NLG2_ActInt_Rx.au8_Data[4];
TempCon_Rx			:=	NLG2_ActInt_Rx.au8_Data[5];
DCHVAhAct_Rx		:=	SHL(USINT_TO_UINT(NLG2_ActInt_Rx.au8_Data[6]), 8) +
								USINT_TO_UINT(NLG2_ActInt_Rx.au8_Data[7]);
(*Act Lim*)
StateCrtlPilot		:=	SHR((NLG2_ActLim_Rx.au8_Data[0] AND 2#11100000), 5);
DCHVVoltAct_Rx	:=	SHL(USINT_TO_UINT(NLG2_ActLim_Rx.au8_Data[0] AND 2#00011111), 8) +
								USINT_TO_UINT(NLG2_ActLim_Rx.au8_Data[1]);
StateAct			:=	SHR((NLG2_ActLim_Rx.au8_Data[2] AND 2#11100000), 5);
S_DCHVCurrLim		:=	NLG2_ActLim_Rx.au8_Data[2].4;
S_DCHVVoltLim		:=	NLG2_ActLim_Rx.au8_Data[2].3;
DCHVCurrAct_Rx	:=	SHL(USINT_TO_UINT(NLG2_ActLim_Rx.au8_Data[2] AND 2#00000111), 8) +
								USINT_TO_UINT(NLG2_ActLim_Rx.au8_Data[3]);
S_ProximityLim		:=	NLG2_ActLim_Rx.au8_Data[4].7;
S_CtrlPilotLim		:=	NLG2_ActLim_Rx.au8_Data[4].6;
S_ConTempLim		:=	NLG2_ActLim_Rx.au8_Data[4].5;
S_IntTempLim		:=	NLG2_ActLim_Rx.au8_Data[4].4;
S_ACCurrLim			:=	NLG2_ActLim_Rx.au8_Data[4].3;
ACCurrMaxAct_Rx	:=	SHL(USINT_TO_UINT(NLG2_ActLim_Rx.au8_Data[4] AND 2#00000111), 8) +
								USINT_TO_UINT(NLG2_ActLim_Rx.au8_Data[5]);
ACCurrHWAvl_Rx		:=	NLG2_ActLim_Rx.au8_Data[6];
S_ProximityDet		:=	NLG2_ActLim_Rx.au8_Data[7].7;
S_CtrlPilotDet		:=	NLG2_ActLim_Rx.au8_Data[7].6;
S_ConLocked			:=	NLG2_ActLim_Rx.au8_Data[7].5;
S_ACDet				:=	NLG2_ActLim_Rx.au8_Data[7].4;
S_HWWakeup			:=	NLG2_ActLim_Rx.au8_Data[7].3;
S_HWEnablErre		:=	NLG2_ActLim_Rx.au8_Data[7].2;
S_Err				:=	NLG2_ActLim_Rx.au8_Data[7].1;
S_Warn				:=	NLG2_ActLim_Rx.au8_Data[7].0;
(*Act Plug*)
StatusCP			:=	SHR((NLG2_ActPlug_Rx.au8_Data[0] AND 2#11100000), 5);
S_CPX1				:=	NLG2_ActPlug_Rx.au8_Data[0].4;
S_CPSCC				:=	NLG2_ActPlug_Rx.au8_Data[0].3;
ACCurrMaxCP_Rx	:=	SHL(USINT_TO_UINT(NLG2_ActPlug_Rx.au8_Data[0] AND 2#00000011), 8) +
								USINT_TO_UINT(NLG2_ActPlug_Rx.au8_Data[1]);
StatusPP			:=	SHR((NLG2_ActPlug_Rx.au8_Data[2] AND 2#01110000), 4);
ACCurrMaxPP		:=	NLG2_ActPlug_Rx.au8_Data[2] AND 2#00001111;
s_ACVoltDerate		:=	NLG2_ActPlug_Rx.au8_Data[4].7;
S_ACDerating		:=	NLG2_ActPlug_Rx.au8_Data[4].6;
ACPhaseUsd			:=	SHR((NLG2_ActPlug_Rx.au8_Data[4] AND 2#00111000), 3);
ACPhaseDet			:=	NLG2_ActPlug_Rx.au8_Data[4] AND 2#00000111;
CoolingRequest		:=	NLG2_ActPlug_Rx.au8_Data[5] AND 2#01111111;
TempCoolPlate_Rx	:=	NLG2_ActPlug_Rx.au8_Data[6];


